// TwinCAT 3 PLC project Untitled1
// Title: B300S
// Company: LS do Brasil
// Author: Thiago Carlos
// ProjectVersion: 1.1
// Description: Programa da máquina B300S, 12 liquidos e dois pós
// ProgramVersion: 3.1.4024.0
// libraries:
//   Tc2_ControllerToolbox, * (Beckhoff Automation GmbH)
//   Tc2_Database, * (Beckhoff Automation GmbH)
//   Tc2_EtherCAT, * (Beckhoff Automation GmbH)
//   Tc2_Standard, * (Beckhoff Automation GmbH)
//   Tc2_System, * (Beckhoff Automation GmbH)
//   Tc2_Utilities, * (Beckhoff Automation GmbH)
//   Tc3_Database, * (Beckhoff Automation GmbH)
//   Tc3_EventLogger, * (Beckhoff Automation GmbH)
//   Tc3_IPCDiag, * (Beckhoff Automation GmbH)
//   Tc3_Module, * (Beckhoff Automation GmbH)
// project tree:
//   DUTs/ DUT_cfgBombas.TcDUT, DUT_cfgPosicValvula.TcDUT, DUT_PosicValvula.TcDUT, RecetaEdicion.TcDUT, stComboBoxRecipes.TcDUT, stListado_Liquidos.TcDUT, stListado_Polvos.TcDUT, stReceta_Circuito.TcDUT, stReceta_Polvo.TcDUT, u_RPM.TcDUT, u_SM6020.TcDUT, u_SM6020_caudal.TcDUT, u_SM6020_temp.TcDUT
//   / GVL.TcGVL, PlcTask.TcTTO
//   GVLs/ CanOpen.TcGVL, Configura.TcGVL, DatosProceso.TcGVL, Entradas.TcGVL, HMI.TcGVL, HMICA1.TcGVL, HMICA2.TcGVL, HMICA3.TcGVL, HMIcalP1.TcGVL, HMIcalP2.TcGVL, ioLink.TcGVL, Liquidos.TcGVL, Polvos.TcGVL, RecetasGestion.TcGVL, Receta_Activa.TcGVL, SafetyInputs.TcGVL, Salidas.TcGVL, Seguridad.TcGVL
//   POUs/ Agitadores.TcPOU, Alarmas.TcPOU, Balanza_Semilla.TcPOU, Datos_Caudalimetros.TcPOU, Datos_Variadores.TcPOU, Inicio.TcPOU, MAIN.TcPOU, PasosDosificar.TcPOU, PrecargaLiqInyeccion.TcPOU, Tabla_FIFO.TcPOU, VarPersistentes.TcPOU, Tratadora.TcPOU, _Seguridad.TcPOU
//   POUs/CanOpen/ SDO_READ.TcPOU
//   POUs/Control Equipos/ ControlValv_ioLink.TcPOU, Equipo_Motor_ATV320.TcPOU, Equipo_Motor_No_Rev.TcPOU, Equipo_Valvula_5_2.TcPOU, Equipo_Valvula_5_2_biestable.TcPOU
//   POUs/Elementos/ Calculo_caudal.TcPOU, Calc_Veloc_Polvo.TcPOU, Calibracion_Liq_calc.TcPOU, Calibracion_Po_calc.TcPOU, CorrecionCaudalxOffset.TcPOU, FB_PID.TcPOU, Tiempo_seg_to_TIME.TcPOU, Tiempo_TIME_to_seg.TcPOU
//   POUs/Lavado/ AbreValvulasLavagem.TcPOU, Valvulas_Lavado.TcPOU
//   POUs/Perifericos/ Carga_semilla.TcPOU, Descarga_semilla.TcPOU
//   POUs/Pesajes/ Balanza.TcPOU
//   POUs/Polvo 1/ Dosificador_Polvo_1.TcPOU
//   POUs/Polvo 2/ Dosificador_Polvo_2.TcPOU
//   POUs/Puesto_Calibracion_1/ Circuito_L1.TcPOU, Circuito_L2.TcPOU, Circuito_L3.TcPOU, Circuito_L4.TcPOU, Puesto_CA1.TcPOU
//   POUs/Puesto_Calibracion_2/ Circuito_L5.TcPOU, Circuito_L6.TcPOU, Circuito_L7.TcPOU, Circuito_L8.TcPOU, Puesto_CA2.TcPOU
//   POUs/Puesto_Calibracion_3/ Circuito_L11.TcPOU, Circuito_L12.TcPOU, Circuito_L9.TcPOU, Circuito_L10.TcPOU, Puesto_CA3.TcPOU
//   POUs/Receitas %28Thiago%29/ Receitas.TcPOU (not stored)
//   POUs/Secuencias/ Porc_inicial_Bomba.TcPOU, Totalizador.TcPOU, VeloAspersorAuto.TcPOU, LavadoCircuitoLiquidos.TcPOU
//   POUs/Testes Thiago/ AlarmesDaMaquina.TcPOU, AquecimentoValvulas.TcPOU, CalculoConsumo.TcPOU, Calibracao_V03.TcPOU, ConfigBombas.TcPOU, ConsumoIBCs.TcPOU, E_State.TcDUT, Filtro.TcPOU, Filtro2.TcPOU, GeraAlarme.TcPOU, BancoDeDados.TcPOU, Calibracao_V02.TcPOU, DUT_ConfigLavagem.TcDUT, DUT_EventLogger.TcDUT, InsertBD_Comandos.TcPOU, IntervaloLavCalibr.TcPOU, iPC_Diagnostic.TcPOU, Lavagem.TcPOU, LiqNaReceita.TcPOU, MediaMovel.TcPOU, Percentual.TcPOU, PRG_DE_TESTES.TcPOU, ST_SelectStruct.TcDUT, Testes.TcGVL, TONR.TcPOU
//   POUs/TestesPID/ PID_GENERICO.TcPOU
// real-time tasks:
//   TASK PlcTask: cycle T#10ms, priority 6, ADS port 352
// I/O:
//   DEVICE Dispositivos (EtherCAT) (disabled), AmsNetId 192.168.10.68.2.1
//     C1 (EK1100) [EK1100 EtherCAT Coupler (2A E-Bus)]
//       C2 (EL6070) [EL6070 1Ch. Licensing-Terminal]
//       C3 (EL1809) [EL1809 16Ch. Dig. Input 24V, 3ms]
//       C4 (EL2809) [EL2809 16Ch. Dig. Output 24V, 0.5A]
//       C6 (EL6224) [EL6224 (IO Link Master)]
//       C5 (EL2911) [EL2911, Potential supply terminal (10 A) with 4 Ch. Safety Inputs, TwinSAFE]
//         modules: Module 2 (FSOUT), Module 3 (DEVICEIO), Module 4 (FSLOGIC)
//       C7 (EL6753) [EL6751 CANopen Master]
//       C8 (EK1122) [EK1122 2 port EtherCAT junction]
//         CA1_1 (ifm IO-Link Master AL1332) [ifm IO-Link Master AL1332]
//           modules: Module 1 (IOL_16/4_I/O-Bytes), Module 2 (IOL_4/4_I/O-Bytes), Module 3 (IOL_16/4_I/O-Bytes), Module 4 (IOL_4/4_I/O-Bytes), Module 5 (IOL_16/4_I/O-Bytes), Module 6 (IOL_4/4_I/O-Bytes), Module 7 (IOL_16/4_I/O-Bytes), Module 8 (IOL_4/4_I/O-Bytes)
//         CA1_2 (EP3356-0022) [EP3356-0022 1Ch. Ana. Input Resistor Bridge Terminal, 24bit, High Precision]
//         PU1_1 (EP3356-0022) [EP3356-0022 1Ch. Ana. Input Resistor Bridge Terminal, 24bit, High Precision]
//         PU1_2 (ifm IO-Link Master AL1332) [ifm IO-Link Master AL1332]
//           modules: Module 1 (IOL_4/4_I/O-Bytes), Module 2 (IOL_4/4_I/O-Bytes), Module 3 (IOL_4/4_I/O-Bytes), Module 4 (IOL_4/4_I/O-Bytes), Module 5 (IOL_4/4_I/O-Bytes), Module 6 (IOL_4/4_I/O-Bytes), Module 7 (Digital_IN), Module 8 (Digital_IN)
//         PU1_3 (EP3356-0022) [EP3356-0022 1Ch. Ana. Input Resistor Bridge Terminal, 24bit, High Precision]
//         PU1_4 (EP3356-0022) [EP3356-0022 1Ch. Ana. Input Resistor Bridge Terminal, 24bit, High Precision]
//         PU1_5 (ifm IO-Link Master AL1332) [ifm IO-Link Master AL1332]
//           modules: Module 1 (IOL_4/4_I/O-Bytes), Module 2 (IOL_4/4_I/O-Bytes), Module 3 (IOL_4/4_I/O-Bytes), Module 4 (IOL_4/4_I/O-Bytes), Module 5 (IOL_4/4_I/O-Bytes), Module 6 (IOL_4/4_I/O-Bytes), Module 7 (Digital_IN), Module 8 (Digital_IN)
//         PU1_6 (EP3356-0022) [EP3356-0022 1Ch. Ana. Input Resistor Bridge Terminal, 24bit, High Precision]
//         PU4_1 (ifm IO-Link Master AL1330) [ifm IO-Link Master AL1330]
//           modules: Module 1 (IOL_4/4_I/O-Bytes), Module 2 (IOL_4/4_I/O-Bytes), Module 3 (IOL_4/4_I/O-Bytes), Module 4 (IOL_4/4_I/O-Bytes)
//         CA2_1 (ifm IO-Link Master AL1332) [ifm IO-Link Master AL1332]
//           modules: Module 1 (IOL_16/4_I/O-Bytes), Module 2 (IOL_4/4_I/O-Bytes), Module 3 (IOL_16/4_I/O-Bytes), Module 4 (IOL_4/4_I/O-Bytes), Module 5 (IOL_16/4_I/O-Bytes), Module 6 (IOL_4/4_I/O-Bytes), Module 7 (IOL_16/4_I/O-Bytes), Module 8 (IOL_4/4_I/O-Bytes)
//         CA2_2 (EP3356-0022) [EP3356-0022 1Ch. Ana. Input Resistor Bridge Terminal, 24bit, High Precision]
//         PU2_1 (EP3356-0022) [EP3356-0022 1Ch. Ana. Input Resistor Bridge Terminal, 24bit, High Precision]
//         PU2_2 (ifm IO-Link Master AL1332) [ifm IO-Link Master AL1332]
//           modules: Module 1 (IOL_4/4_I/O-Bytes), Module 2 (IOL_4/4_I/O-Bytes), Module 3 (IOL_4/4_I/O-Bytes), Module 4 (IOL_4/4_I/O-Bytes), Module 5 (IOL_4/4_I/O-Bytes), Module 6 (IOL_4/4_I/O-Bytes), Module 7 (Digital_IN), Module 8 (Digital_IN)
//         PU2_3 (EP3356-0022) [EP3356-0022 1Ch. Ana. Input Resistor Bridge Terminal, 24bit, High Precision]
//         PU2_4 (EP3356-0022) [EP3356-0022 1Ch. Ana. Input Resistor Bridge Terminal, 24bit, High Precision]
//         PU2_5 (ifm IO-Link Master AL1332) [ifm IO-Link Master AL1332]
//           modules: Module 1 (IOL_4/4_I/O-Bytes), Module 2 (IOL_4/4_I/O-Bytes), Module 3 (IOL_4/4_I/O-Bytes), Module 4 (IOL_4/4_I/O-Bytes), Module 5 (IOL_4/4_I/O-Bytes), Module 6 (IOL_4/4_I/O-Bytes), Module 7 (Digital_IN), Module 8 (Digital_IN)
//         PU2_6 (EP3356-0022) [EP3356-0022 1Ch. Ana. Input Resistor Bridge Terminal, 24bit, High Precision]
//       C9 (EK1122) [EK1122 2 port EtherCAT junction]
//         CA3_1 (ifm IO-Link Master AL1332) [ifm IO-Link Master AL1332]
//           modules: Module 1 (IOL_16/4_I/O-Bytes), Module 2 (IOL_4/4_I/O-Bytes), Module 3 (IOL_16/4_I/O-Bytes), Module 4 (IOL_4/4_I/O-Bytes), Module 5 (IOL_16/4_I/O-Bytes), Module 6 (IOL_4/4_I/O-Bytes), Module 7 (IOL_16/4_I/O-Bytes), Module 8 (IOL_4/4_I/O-Bytes)
//         CA3_2 (EP3356-0022) [EP3356-0022 1Ch. Ana. Input Resistor Bridge Terminal, 24bit, High Precision]
//         PU3_1 (EP3356-0022) [EP3356-0022 1Ch. Ana. Input Resistor Bridge Terminal, 24bit, High Precision]
//         PU3_2 (ifm IO-Link Master AL1332) [ifm IO-Link Master AL1332]
//           modules: Module 1 (IOL_4/4_I/O-Bytes), Module 2 (IOL_4/4_I/O-Bytes), Module 3 (IOL_4/4_I/O-Bytes), Module 4 (IOL_4/4_I/O-Bytes), Module 5 (IOL_4/4_I/O-Bytes), Module 6 (IOL_4/4_I/O-Bytes), Module 7 (Digital_IN), Module 8 (Digital_IN)
//         PU3_3 (EP3356-0022) [EP3356-0022 1Ch. Ana. Input Resistor Bridge Terminal, 24bit, High Precision]
//         PU3_4 (EP3356-0022) [EP3356-0022 1Ch. Ana. Input Resistor Bridge Terminal, 24bit, High Precision]
//         PU3_5 (ifm IO-Link Master AL1332) [ifm IO-Link Master AL1332]
//           modules: Module 1 (IOL_4/4_I/O-Bytes), Module 2 (IOL_4/4_I/O-Bytes), Module 3 (IOL_4/4_I/O-Bytes), Module 4 (IOL_4/4_I/O-Bytes), Module 5 (IOL_4/4_I/O-Bytes), Module 6 (IOL_4/4_I/O-Bytes), Module 7 (Digital_IN), Module 8 (Digital_IN)
//         PU3_6 (EP3356-0022) [EP3356-0022 1Ch. Ana. Input Resistor Bridge Terminal, 24bit, High Precision]
//         PE_2 (ifm IO-Link Master AL1332) [ifm IO-Link Master AL1332]
//           modules: Module 1 (IOL_4/4_I/O-Bytes), Module 2 (IOL_4/4_I/O-Bytes), Module 3 (IOL_4/4_I/O-Bytes), Module 4 (IOL_4/4_I/O-Bytes), Module 5 (IOL_4/4_I/O-Bytes), Module 6 (IOL_4/4_I/O-Bytes), Module 7 (IOL_4/4_I/O-Bytes), Module 8 (IOL_4/4_I/O-Bytes)
//         PE_1 (EX260-SEC1) [EX260-SEC1 EtherCAT SI Unit (32DO_PNP) Rev1.2]
//         PE_4 (ifm IO-Link Master AL1330) [ifm IO-Link Master AL1330]
//           modules: Module 1 (IOL_4/4_I/O-Bytes), Module 2 (Digital_IN), Module 3 (Digital_IN), Module 4 (Digital_IN)
//         PE_3 (EX260-SEC1) [EX260-SEC1 EtherCAT SI Unit (32DO_PNP) Rev1.2]
//         Box 37 (EX260-SEC1) [EX260-SEC1 EtherCAT SI Unit (32DO_PNP) Rev1.2] (disabled)
//     TR_1 (EP3356-0022) [EP3356-0022 1Ch. Ana. Input Resistor Bridge Terminal, 24bit, High Precision]
//     TR_2 (EP1908) [EP1908, 8 Ch. Safety Input 24V, TwinSAFE ]
//       modules: Module 1 (FSOE)
//     TR_3 (EP1908) [EP1908, 8 Ch. Safety Input 24V, TwinSAFE ]
//       modules: Module 1 (FSOE)
//     TR_4 (ifm IO-Link Master AL1332) [ifm IO-Link Master AL1332]
//       modules: Module 1 (Digital_IN), Module 2 (Digital_IN), Module 3 (Digital_IN), Module 4 (Digital_IN), Module 5 (Digital_IN), Module 6 (Digital_IN), Module 7 (IOL_In_4Byte), Module 8 (IOL_In_4Byte)
//     TR_5 (EX260-SEC1) [EX260-SEC1 EtherCAT SI Unit (32DO_PNP) Rev1.2]
//     TR_6 (ifm IO-Link Master AL1332) [ifm IO-Link Master AL1332]
//       modules: Module 1 (IOL_16/4_I/O-Bytes), Module 2 (IOL_16/4_I/O-Bytes), Module 3 (IOL_16/4_I/O-Bytes), Module 4 (IOL_16/4_I/O-Bytes), Module 5 (IOL_16/4_I/O-Bytes), Module 6 (IOL_16/4_I/O-Bytes), Module 7 (IOL_16/4_I/O-Bytes), Module 8 (IOL_16/4_I/O-Bytes)
//     TR_7 (ifm IO-Link Master AL1330) [ifm IO-Link Master AL1330]
//       modules: Module 1 (IOL_16/4_I/O-Bytes), Module 2 (IOL_16/4_I/O-Bytes), Module 3 (IOL_16/4_I/O-Bytes), Module 4 (IOL_16/4_I/O-Bytes)
//     TR_8 (ifm IO-Link Master AL1332) [ifm IO-Link Master AL1332]
//       modules: Module 1 (IOL_4/4_I/O-Bytes), Module 2 (IOL_4/4_I/O-Bytes), Module 3 (Digital_IN), Module 4 (Digital_IN), Module 5 (Digital_IN), Module 6 (Digital_OUT), Module 7 (IOL_4/4_I/O-Bytes), Module 8 (IOL_4/4_I/O-Bytes)
//     TR_9 (ifm IO-Link Master AL1330) [ifm IO-Link Master AL1330]
//       modules: Module 1 (Digital_IN), Module 2 (Digital_IN), Module 3 (Digital_IN), Module 4 (IOL_4/4_I/O-Bytes)
//     TR_10 (EP3356-0022) [EP3356-0022 1Ch. Ana. Input Resistor Bridge Terminal, 24bit, High Precision]
//     TR_11 (ifm IO-Link Master AL1330) [ifm IO-Link Master AL1330]
//       modules: Module 1 (Digital_IN), Module 2 (Digital_IN), Module 3 (Digital_IN), Module 4 (Digital_IN)
//     TR_12 (EP3356-0022) [EP3356-0022 1Ch. Ana. Input Resistor Bridge Terminal, 24bit, High Precision]
//   DEVICE Device 2 (EL6751), AmsNetId 169.254.25.50.4.1
//     Box 1 (ATV320D15N4C)
//     Box 2 (ATV320U07M2C)
//     Box 3 (ATV320U06M2C)
//     Box 4 (ATV320U06M2C)
//     Box 5 (ATV320U07M2C)
//     Box 6 (ATV320U04M2C)
//     Box 7 (ATV320U04M2C)
//     Box 8 (ATV320U04M2C)
//     Box 9 (ATV320U04M2C)
//     Box 10 (ATV320U04M2C)
//     Box 11 (ATV320U04M2C)
//     Box 12 (ATV320U04M2C)
//     Box 13 (ATV320U04M2C)
//     Box 14 (ATV320U04M2C)
//     Box 15 (ATV320U04M2C)
//     Box 16 (ATV320U04M2C)
//     Box 17 (ATV320U15M2C)
//     Box 18 (ATV320U15M2C)
//     Box 19 (ATV320U22M2C)
//     Box 34 (ATV320U04M2C)
//     Box 35 (ATV320U04M2C)
// variable links:
//   Dispositivos (EtherCAT) <-> Dispositivos (EtherCAT)/C1 (EK1100)/C5 (EL2911)
//     TR_2 (EP1908)/Module 1 (FSOE)/FSOE Outputs/FSOE <-> ConnectionInputs/Message_18 TxPDO
//   Dispositivos (EtherCAT) <-> Dispositivos (EtherCAT)/TR_2 (EP1908)
//     C1 (EK1100)/C5 (EL2911)/ConnectionOutputs/Message_18 RxPDO <-> Module 1 (FSOE)/FSOE Inputs/FSOE
//   Dispositivos (EtherCAT) <-> Dispositivos (EtherCAT)/TR_3 (EP1908)
//     C1 (EK1100)/C5 (EL2911)/ConnectionInputs/Message_19 TxPDO <-> Module 1 (FSOE)/FSOE Outputs/FSOE
//     C1 (EK1100)/C5 (EL2911)/ConnectionOutputs/Message_19 RxPDO <-> Module 1 (FSOE)/FSOE Inputs/FSOE
//   Untitled1/Untitled1 Instance <-> Device 2 (EL6751)/Box 1 (ATV320D15N4C)
//     PlcTask Inputs/Entradas.wTR_S_VF1_PV <-> TxPDO 1/Inputs/VarIn-1
//     PlcTask Inputs/Entradas.wTR_S_VF1_St <-> TxPDO 1/Inputs/VarIn-0
//     PlcTask Outputs/Salidas.wTR_S_VF1_Cmd <-> RxPDO 1/Outputs/VarOut-0
//     PlcTask Outputs/Salidas.wTR_S_VF1_Set <-> RxPDO 1/Outputs/VarOut-1
//   Untitled1/Untitled1 Instance <-> Device 2 (EL6751)/Box 10 (ATV320U04M2C)
//     PlcTask Inputs/Entradas.wPP2_L6_BD_PV <-> TxPDO 1/Inputs/VarIn-1
//     PlcTask Inputs/Entradas.wPP2_L6_BD_St <-> TxPDO 1/Inputs/VarIn-0
//     PlcTask Outputs/Salidas.wPP2_L6_BD_Cmd <-> RxPDO 1/Outputs/VarOut-0
//     PlcTask Outputs/Salidas.wPP2_L6_BD_Set <-> RxPDO 1/Outputs/VarOut-1
//   Untitled1/Untitled1 Instance <-> Device 2 (EL6751)/Box 11 (ATV320U04M2C)
//     PlcTask Inputs/Entradas.wPP2_L7_BD_PV <-> TxPDO 1/Inputs/VarIn-1
//     PlcTask Inputs/Entradas.wPP2_L7_BD_St <-> TxPDO 1/Inputs/VarIn-0
//     PlcTask Outputs/Salidas.wPP2_L7_BD_Cmd <-> RxPDO 1/Outputs/VarOut-0
//     PlcTask Outputs/Salidas.wPP2_L7_BD_Set <-> RxPDO 1/Outputs/VarOut-1
//   Untitled1/Untitled1 Instance <-> Device 2 (EL6751)/Box 12 (ATV320U04M2C)
//     PlcTask Inputs/Entradas.wPP2_L8_BD_PV <-> TxPDO 1/Inputs/VarIn-1
//     PlcTask Inputs/Entradas.wPP2_L8_BD_St <-> TxPDO 1/Inputs/VarIn-0
//     PlcTask Outputs/Salidas.wPP2_L8_BD_Cmd <-> RxPDO 1/Outputs/VarOut-0
//     PlcTask Outputs/Salidas.wPP2_L8_BD_Set <-> RxPDO 1/Outputs/VarOut-1
//   Untitled1/Untitled1 Instance <-> Device 2 (EL6751)/Box 13 (ATV320U04M2C)
//     PlcTask Inputs/Entradas.wPP3_L9_BD_PV <-> TxPDO 1/Inputs/VarIn-1
//     PlcTask Inputs/Entradas.wPP3_L9_BD_St <-> TxPDO 1/Inputs/VarIn-0
//     PlcTask Outputs/Salidas.wPP3_L9_BD_Cmd <-> RxPDO 1/Outputs/VarOut-0
//     PlcTask Outputs/Salidas.wPP3_L9_BD_Set <-> RxPDO 1/Outputs/VarOut-1
//   Untitled1/Untitled1 Instance <-> Device 2 (EL6751)/Box 14 (ATV320U04M2C)
//     PlcTask Inputs/Entradas.wPP3_L10_BD_PV <-> TxPDO 1/Inputs/VarIn-1
//     PlcTask Inputs/Entradas.wPP3_L10_BD_St <-> TxPDO 1/Inputs/VarIn-0
//     PlcTask Outputs/Salidas.wPP3_L10_BD_Cmd <-> RxPDO 1/Outputs/VarOut-0
//     PlcTask Outputs/Salidas.wPP3_L10_BD_Set <-> RxPDO 1/Outputs/VarOut-1
//   Untitled1/Untitled1 Instance <-> Device 2 (EL6751)/Box 15 (ATV320U04M2C)
//     PlcTask Inputs/Entradas.wPP3_L11_BD_PV <-> TxPDO 1/Inputs/VarIn-1
//     PlcTask Inputs/Entradas.wPP3_L11_BD_St <-> TxPDO 1/Inputs/VarIn-0
//     PlcTask Outputs/Salidas.wPP3_L11_BD_Cmd <-> RxPDO 1/Outputs/VarOut-0
//     PlcTask Outputs/Salidas.wPP3_L11_BD_Set <-> RxPDO 1/Outputs/VarOut-1
//   Untitled1/Untitled1 Instance <-> Device 2 (EL6751)/Box 16 (ATV320U04M2C)
//     PlcTask Inputs/Entradas.wPP3_L12_BD_PV <-> TxPDO 1/Inputs/VarIn-1
//     PlcTask Inputs/Entradas.wPP3_L12_BD_St <-> TxPDO 1/Inputs/VarIn-0
//     PlcTask Outputs/Salidas.wPP3_L12_BD_Cmd <-> RxPDO 1/Outputs/VarOut-0
//     PlcTask Outputs/Salidas.wPP3_L12_BD_Set <-> RxPDO 1/Outputs/VarOut-1
//   Untitled1/Untitled1 Instance <-> Device 2 (EL6751)/Box 17 (ATV320U15M2C)
//     PlcTask Inputs/Entradas.wPE_H_VF1_PV <-> TxPDO 1/Inputs/VarIn-1
//     PlcTask Inputs/Entradas.wPE_H_VF1_St <-> TxPDO 1/Inputs/VarIn-0
//     PlcTask Outputs/Salidas.wPE_H_VF1_Cmd <-> RxPDO 1/Outputs/VarOut-0
//     PlcTask Outputs/Salidas.wPE_H_VF1_Set <-> RxPDO 1/Outputs/VarOut-1
//   Untitled1/Untitled1 Instance <-> Device 2 (EL6751)/Box 18 (ATV320U15M2C)
//     PlcTask Inputs/Entradas.wPE_H_VF2_PV <-> TxPDO 1/Inputs/VarIn-1
//     PlcTask Inputs/Entradas.wPE_H_VF2_St <-> TxPDO 1/Inputs/VarIn-0
//     PlcTask Outputs/Salidas.wPE_H_VF2_Cmd <-> RxPDO 1/Outputs/VarOut-0
//     PlcTask Outputs/Salidas.wPE_H_VF2_Set <-> RxPDO 1/Outputs/VarOut-1
//   Untitled1/Untitled1 Instance <-> Device 2 (EL6751)/Box 19 (ATV320U22M2C)
//     PlcTask Inputs/Entradas.wPE_B_VF1_PV <-> TxPDO 1/Inputs/VarIn-1
//     PlcTask Inputs/Entradas.wPE_B_VF1_St <-> TxPDO 1/Inputs/VarIn-0
//     PlcTask Outputs/Salidas.wPE_B_VF1_Cmd <-> RxPDO 1/Outputs/VarOut-0
//     PlcTask Outputs/Salidas.wPE_B_VF1_Set <-> RxPDO 1/Outputs/VarOut-1
//   Untitled1/Untitled1 Instance <-> Device 2 (EL6751)/Box 2 (ATV320U07M2C)
//     PlcTask Inputs/Entradas.wTR_S_VF2_PV <-> TxPDO 1/Inputs/VarIn-1
//     PlcTask Inputs/Entradas.wTR_S_VF2_St <-> TxPDO 1/Inputs/VarIn-0
//     PlcTask Outputs/Salidas.wTR_S_VF2_Cmd <-> RxPDO 1/Outputs/VarOut-0
//     PlcTask Outputs/Salidas.wTR_S_VF2_Set <-> RxPDO 1/Outputs/VarOut-1
//   Untitled1/Untitled1 Instance <-> Device 2 (EL6751)/Box 3 (ATV320U06M2C)
//     PlcTask Inputs/Entradas.TR_P1_VF_PV <-> TxPDO 1/Inputs/VarIn-1
//     PlcTask Inputs/Entradas.TR_P1_VF_St <-> TxPDO 1/Inputs/VarIn-0
//     PlcTask Outputs/Salidas.TR_P1_VF_Cmd <-> RxPDO 1/Outputs/VarOut-0
//     PlcTask Outputs/Salidas.TR_P1_VF_Set <-> RxPDO 1/Outputs/VarOut-1
//   Untitled1/Untitled1 Instance <-> Device 2 (EL6751)/Box 34 (ATV320U04M2C)
//     PlcTask Inputs/Entradas.TR_P1_VI_PV <-> TxPDO 1/Inputs/VarIn-1
//     PlcTask Inputs/Entradas.TR_P1_VI_St <-> TxPDO 1/Inputs/VarIn-0
//     PlcTask Outputs/Salidas.TR_P1_VI_Cmd <-> RxPDO 1/Outputs/VarOut-0
//     PlcTask Outputs/Salidas.TR_P1_VI_Set <-> RxPDO 1/Outputs/VarOut-1
//   Untitled1/Untitled1 Instance <-> Device 2 (EL6751)/Box 35 (ATV320U04M2C)
//     PlcTask Inputs/Entradas.TR_P2_VI_PV <-> TxPDO 1/Inputs/VarIn-1
//     PlcTask Inputs/Entradas.TR_P2_VI_St <-> TxPDO 1/Inputs/VarIn-0
//     PlcTask Outputs/Salidas.TR_P2_VI_Cmd <-> RxPDO 1/Outputs/VarOut-0
//     PlcTask Outputs/Salidas.TR_P2_VI_Set <-> RxPDO 1/Outputs/VarOut-1
//   Untitled1/Untitled1 Instance <-> Device 2 (EL6751)/Box 4 (ATV320U06M2C)
//     PlcTask Inputs/Entradas.TR_P2_VF_PV <-> TxPDO 1/Inputs/VarIn-1
//     PlcTask Inputs/Entradas.TR_P2_VF_St <-> TxPDO 1/Inputs/VarIn-0
//     PlcTask Outputs/Salidas.TR_P2_VF_Cmd <-> RxPDO 1/Outputs/VarOut-0
//     PlcTask Outputs/Salidas.TR_P2_VF_Set <-> RxPDO 1/Outputs/VarOut-1
//   Untitled1/Untitled1 Instance <-> Device 2 (EL6751)/Box 5 (ATV320U07M2C)
//     PlcTask Inputs/Entradas.wPP1_L1_BD_PV <-> TxPDO 1/Inputs/VarIn-1
//     PlcTask Inputs/Entradas.wPP1_L1_BD_St <-> TxPDO 1/Inputs/VarIn-0
//     PlcTask Outputs/Salidas.wPP1_L1_BD_Cmd <-> RxPDO 1/Outputs/VarOut-0
//     PlcTask Outputs/Salidas.wPP1_L1_BD_Set <-> RxPDO 1/Outputs/VarOut-1
//   Untitled1/Untitled1 Instance <-> Device 2 (EL6751)/Box 6 (ATV320U04M2C)
//     PlcTask Inputs/Entradas.wPP1_L2_BD_PV <-> TxPDO 1/Inputs/VarIn-1
//     PlcTask Inputs/Entradas.wPP1_L2_BD_St <-> TxPDO 1/Inputs/VarIn-0
//     PlcTask Outputs/Salidas.wPP1_L2_BD_Cmd <-> RxPDO 1/Outputs/VarOut-0
//     PlcTask Outputs/Salidas.wPP1_L2_BD_Set <-> RxPDO 1/Outputs/VarOut-1
//   Untitled1/Untitled1 Instance <-> Device 2 (EL6751)/Box 7 (ATV320U04M2C)
//     PlcTask Inputs/Entradas.wPP1_L3_BD_PV <-> TxPDO 1/Inputs/VarIn-1
//     PlcTask Inputs/Entradas.wPP1_L3_BD_St <-> TxPDO 1/Inputs/VarIn-0
//     PlcTask Outputs/Salidas.wPP1_L3_BD_Cmd <-> RxPDO 1/Outputs/VarOut-0
//     PlcTask Outputs/Salidas.wPP1_L3_BD_Set <-> RxPDO 1/Outputs/VarOut-1
//   Untitled1/Untitled1 Instance <-> Device 2 (EL6751)/Box 8 (ATV320U04M2C)
//     PlcTask Inputs/Entradas.wPP1_L4_BD_PV <-> TxPDO 1/Inputs/VarIn-1
//     PlcTask Inputs/Entradas.wPP1_L4_BD_St <-> TxPDO 1/Inputs/VarIn-0
//     PlcTask Outputs/Salidas.wPP1_L4_BD_Cmd <-> RxPDO 1/Outputs/VarOut-0
//     PlcTask Outputs/Salidas.wPP1_L4_BD_Set <-> RxPDO 1/Outputs/VarOut-1
//   Untitled1/Untitled1 Instance <-> Device 2 (EL6751)/Box 9 (ATV320U04M2C)
//     PlcTask Inputs/Entradas.wPP2_L5_BD_PV <-> TxPDO 1/Inputs/VarIn-1
//     PlcTask Inputs/Entradas.wPP2_L5_BD_St <-> TxPDO 1/Inputs/VarIn-0
//     PlcTask Outputs/Salidas.wPP2_L5_BD_Cmd <-> RxPDO 1/Outputs/VarOut-0
//     PlcTask Outputs/Salidas.wPP2_L5_BD_Set <-> RxPDO 1/Outputs/VarOut-1
//   Untitled1/Untitled1 Instance <-> Dispositivos (EtherCAT)/C1 (EK1100)/C3 (EL1809)
//     PlcTask Inputs/Entradas.ReposicionEmerg <-> Channel 15/Input
//     PlcTask Inputs/Entradas.bPP1_L1_AG_Z <-> Channel 2/Input
//     PlcTask Inputs/Entradas.bPP1_L2_AG_Z <-> Channel 3/Input
//     PlcTask Inputs/Entradas.bPP1_L3_AG_Z <-> Channel 4/Input
//     PlcTask Inputs/Entradas.bPP1_L4_AG_Z <-> Channel 5/Input
//     PlcTask Inputs/Entradas.bPP2_L5_AG_Z <-> Channel 6/Input
//     PlcTask Inputs/Entradas.bPP2_L6_AG_Z <-> Channel 7/Input
//     PlcTask Inputs/Entradas.bPP2_L7_AG_Z <-> Channel 8/Input
//     PlcTask Inputs/Entradas.bPP2_L8_AG_Z <-> Channel 9/Input
//     PlcTask Inputs/Entradas.bPP3_L10_AG_Z <-> Channel 11/Input
//     PlcTask Inputs/Entradas.bPP3_L11_AG_Z <-> Channel 12/Input
//     PlcTask Inputs/Entradas.bPP3_L12_AG_Z <-> Channel 13/Input
//     PlcTask Inputs/Entradas.bPP3_L9_AG_Z <-> Channel 10/Input
//     PlcTask Inputs/Entradas.bTR_S_VE1_Z <-> Channel 1/Input
//   Untitled1/Untitled1 Instance <-> Dispositivos (EtherCAT)/C1 (EK1100)/C4 (EL2809)
//     PlcTask Outputs/Salidas.PE_P1_HC <-> Channel 14/Output
//     PlcTask Outputs/Salidas.PE_P2_HC <-> Channel 16/Output
//     PlcTask Outputs/Salidas.bPP1_L1_AG_M <-> Channel 2/Output
//     PlcTask Outputs/Salidas.bPP1_L2_AG_M <-> Channel 3/Output
//     PlcTask Outputs/Salidas.bPP1_L3_AG_M <-> Channel 4/Output
//     PlcTask Outputs/Salidas.bPP1_L4_AG_M <-> Channel 5/Output
//     PlcTask Outputs/Salidas.bPP2_L5_AG_M <-> Channel 6/Output
//     PlcTask Outputs/Salidas.bPP2_L6_AG_M <-> Channel 7/Output
//     PlcTask Outputs/Salidas.bPP2_L7_AG_M <-> Channel 8/Output
//     PlcTask Outputs/Salidas.bPP2_L8_AG_M <-> Channel 9/Output
//     PlcTask Outputs/Salidas.bPP3_L10_AG_M <-> Channel 11/Output
//     PlcTask Outputs/Salidas.bPP3_L11_AG_M <-> Channel 12/Output
//     PlcTask Outputs/Salidas.bPP3_L12_AG_M <-> Channel 13/Output
//     PlcTask Outputs/Salidas.bPP3_L9_AG_M <-> Channel 10/Output
//     PlcTask Outputs/Salidas.bTR_S_VE1 <-> Channel 1/Output
//   Untitled1/Untitled1 Instance <-> Dispositivos (EtherCAT)/C1 (EK1100)/C5 (EL2911)
//     PlcTask Inputs/Seguridad.PB_Emergencia <-> StandardInputs/Standard Out Var 8
//     PlcTask Inputs/Seguridad.ParadaDePorta <-> StandardInputs/Standard Out Var 12
//     PlcTask Outputs/Seguridad.ErrorAck <-> StandardOutputs/Standard In Var 1
//     PlcTask Outputs/Seguridad.ResetPorta <-> StandardOutputs/Standard In Var 14
//     PlcTask Outputs/Seguridad.Restart <-> StandardOutputs/Standard In Var 4
//     PlcTask Outputs/Seguridad.Run <-> StandardOutputs/Standard In Var 2
//   Untitled1/Untitled1 Instance <-> Dispositivos (EtherCAT)/C1 (EK1100)/C8 (EK1122)/CA1_1 (ifm IO-Link Master AL1332)
//     PlcTask Inputs/Entradas.CA1_L1_FT1_caudal/caudal[0] <-> Module 1 (IOL_16/4_I/O-Bytes)/TxPDO/input byte 5
//     PlcTask Inputs/Entradas.CA1_L1_FT1_caudal/caudal[1] <-> Module 1 (IOL_16/4_I/O-Bytes)/TxPDO/input byte 4
//     PlcTask Inputs/Entradas.CA1_L2_FT1_caudal/caudal[0] <-> Module 3 (IOL_16/4_I/O-Bytes)/TxPDO/input byte 5
//     PlcTask Inputs/Entradas.CA1_L2_FT1_caudal/caudal[1] <-> Module 3 (IOL_16/4_I/O-Bytes)/TxPDO/input byte 4
//     PlcTask Inputs/Entradas.CA1_L3_FT1_caudal/caudal[0] <-> Module 5 (IOL_16/4_I/O-Bytes)/TxPDO/input byte 5
//     PlcTask Inputs/Entradas.CA1_L3_FT1_caudal/caudal[1] <-> Module 5 (IOL_16/4_I/O-Bytes)/TxPDO/input byte 4
//     PlcTask Inputs/Entradas.CA1_L4_FT1_caudal/caudal[0] <-> Module 7 (IOL_16/4_I/O-Bytes)/TxPDO/input byte 5
//     PlcTask Inputs/Entradas.CA1_L4_FT1_caudal/caudal[1] <-> Module 7 (IOL_16/4_I/O-Bytes)/TxPDO/input byte 4
//     PlcTask Inputs/Entradas.CA1_L1_FT1_temp/temp[0] <-> Module 1 (IOL_16/4_I/O-Bytes)/TxPDO/input byte 9
//     PlcTask Inputs/Entradas.CA1_L1_FT1_temp/temp[1] <-> Module 1 (IOL_16/4_I/O-Bytes)/TxPDO/input byte 8
//     PlcTask Inputs/Entradas.CA1_L2_FT1_temp/temp[0] <-> Module 3 (IOL_16/4_I/O-Bytes)/TxPDO/input byte 9
//     PlcTask Inputs/Entradas.CA1_L2_FT1_temp/temp[1] <-> Module 3 (IOL_16/4_I/O-Bytes)/TxPDO/input byte 8
//     PlcTask Inputs/Entradas.CA1_L3_FT1_temp/temp[0] <-> Module 5 (IOL_16/4_I/O-Bytes)/TxPDO/input byte 9
//     PlcTask Inputs/Entradas.CA1_L3_FT1_temp/temp[1] <-> Module 5 (IOL_16/4_I/O-Bytes)/TxPDO/input byte 8
//     PlcTask Inputs/Entradas.CA1_L4_FT1_temp/temp[0] <-> Module 7 (IOL_16/4_I/O-Bytes)/TxPDO/input byte 9
//     PlcTask Inputs/Entradas.CA1_L4_FT1_temp/temp[1] <-> Module 7 (IOL_16/4_I/O-Bytes)/TxPDO/input byte 8
//     PlcTask Inputs/Entradas.CA1_L1_FT1_tot/total[0] <-> Module 1 (IOL_16/4_I/O-Bytes)/TxPDO/input byte 3
//     PlcTask Inputs/Entradas.CA1_L1_FT1_tot/total[1] <-> Module 1 (IOL_16/4_I/O-Bytes)/TxPDO/input byte 2
//     PlcTask Inputs/Entradas.CA1_L1_FT1_tot/total[2] <-> Module 1 (IOL_16/4_I/O-Bytes)/TxPDO/input byte 1
//     PlcTask Inputs/Entradas.CA1_L1_FT1_tot/total[3] <-> Module 1 (IOL_16/4_I/O-Bytes)/TxPDO/input byte 0
//     PlcTask Inputs/Entradas.CA1_L2_FT1_tot/total[0] <-> Module 3 (IOL_16/4_I/O-Bytes)/TxPDO/input byte 3
//     PlcTask Inputs/Entradas.CA1_L2_FT1_tot/total[1] <-> Module 3 (IOL_16/4_I/O-Bytes)/TxPDO/input byte 2
//     PlcTask Inputs/Entradas.CA1_L2_FT1_tot/total[2] <-> Module 3 (IOL_16/4_I/O-Bytes)/TxPDO/input byte 1
//     PlcTask Inputs/Entradas.CA1_L2_FT1_tot/total[3] <-> Module 3 (IOL_16/4_I/O-Bytes)/TxPDO/input byte 0
//     PlcTask Inputs/Entradas.CA1_L4_FT1_tot/total[0] <-> Module 7 (IOL_16/4_I/O-Bytes)/TxPDO/input byte 3
//     PlcTask Inputs/Entradas.CA1_L4_FT1_tot/total[1] <-> Module 7 (IOL_16/4_I/O-Bytes)/TxPDO/input byte 2
//     PlcTask Inputs/Entradas.CA1_L4_FT1_tot/total[2] <-> Module 7 (IOL_16/4_I/O-Bytes)/TxPDO/input byte 1
//     PlcTask Inputs/Entradas.CA1_L4_FT1_tot/total[3] <-> Module 7 (IOL_16/4_I/O-Bytes)/TxPDO/input byte 0
//     PlcTask Inputs/Entradas.CA1_L1_V1_POSIC/Posicao[0] <-> Module 2 (IOL_4/4_I/O-Bytes)/TxPDO/input byte 0
//     PlcTask Inputs/Entradas.CA1_L1_V1_POSIC/Posicao[1] <-> Module 2 (IOL_4/4_I/O-Bytes)/TxPDO/input byte 1
//     PlcTask Inputs/Entradas.CA1_L2_V1_POSIC/Posicao[0] <-> Module 4 (IOL_4/4_I/O-Bytes)/TxPDO/input byte 0
//     PlcTask Inputs/Entradas.CA1_L2_V1_POSIC/Posicao[1] <-> Module 4 (IOL_4/4_I/O-Bytes)/TxPDO/input byte 1
//     PlcTask Inputs/Entradas.CA1_L3_V1_POSIC/Posicao[0] <-> Module 6 (IOL_4/4_I/O-Bytes)/TxPDO/input byte 0
//     PlcTask Inputs/Entradas.CA1_L3_V1_POSIC/Posicao[1] <-> Module 6 (IOL_4/4_I/O-Bytes)/TxPDO/input byte 1
//     PlcTask Inputs/Entradas.CA1_L4_V1_POSIC/Posicao[0] <-> Module 8 (IOL_4/4_I/O-Bytes)/TxPDO/input byte 0
//     PlcTask Inputs/Entradas.CA1_L4_V1_POSIC/Posicao[1] <-> Module 8 (IOL_4/4_I/O-Bytes)/TxPDO/input byte 1
//     PlcTask Inputs/Entradas.CA1_L3_FT1_Tot/total[{0..3}] <-> Module 5 (IOL_16/4_I/O-Bytes)/TxPDO/input byte {3..0}  (4 links)
//     PlcTask Inputs/ioLink.b3St1_CA1_L{1..4}_V1 <-> Module {2..8 step 2} (IOL_4/4_I/O-Bytes)/TxPDO/input byte 3  (4 links)
//     PlcTask Outputs/ioLink.b0Cmd_CA1_L{1..4}_V1 <-> Module {2..8 step 2} (IOL_4/4_I/O-Bytes)/RxPDO/output byte 0  (4 links)
//   Untitled1/Untitled1 Instance <-> Dispositivos (EtherCAT)/C1 (EK1100)/C8 (EK1122)/CA1_2 (EP3356-0022)
//     PlcTask Inputs/Entradas.CA1_WT1_bWcState <-> WcState/WcState
//     PlcTask Inputs/Entradas.CA1_WT1_rValue_REAL <-> RMB Value (Real)/Value (Real)
//     PlcTask Inputs/Entradas.CA1_WT1_stEcSlaveAmsNetAdr <-> InfoData/AdsAddr
//     PlcTask Inputs/Entradas.CA1_WT1_wState <-> InfoData/State
//     PlcTask Inputs/Entradas.CA1_WT1_wStatus <-> RMB Status/Status
//     PlcTask Outputs/Salidas.CA1_WT1_wControl <-> RMB Control/Ctrl
//   Untitled1/Untitled1 Instance <-> Dispositivos (EtherCAT)/C1 (EK1100)/C8 (EK1122)/CA2_1 (ifm IO-Link Master AL1332)
//     PlcTask Inputs/Entradas.CA2_L5_FT1_caudal/caudal[0] <-> Module 1 (IOL_16/4_I/O-Bytes)/TxPDO/input byte 5
//     PlcTask Inputs/Entradas.CA2_L5_FT1_caudal/caudal[1] <-> Module 1 (IOL_16/4_I/O-Bytes)/TxPDO/input byte 4
//     PlcTask Inputs/Entradas.CA2_L6_FT1_caudal/caudal[0] <-> Module 3 (IOL_16/4_I/O-Bytes)/TxPDO/input byte 5
//     PlcTask Inputs/Entradas.CA2_L6_FT1_caudal/caudal[1] <-> Module 3 (IOL_16/4_I/O-Bytes)/TxPDO/input byte 4
//     PlcTask Inputs/Entradas.CA2_L7_FT1_caudal/caudal[0] <-> Module 5 (IOL_16/4_I/O-Bytes)/TxPDO/input byte 5
//     PlcTask Inputs/Entradas.CA2_L7_FT1_caudal/caudal[1] <-> Module 5 (IOL_16/4_I/O-Bytes)/TxPDO/input byte 4
//     PlcTask Inputs/Entradas.CA2_L8_FT1_caudal/caudal[0] <-> Module 7 (IOL_16/4_I/O-Bytes)/TxPDO/input byte 5
//     PlcTask Inputs/Entradas.CA2_L8_FT1_caudal/caudal[1] <-> Module 7 (IOL_16/4_I/O-Bytes)/TxPDO/input byte 4
//     PlcTask Inputs/Entradas.CA2_L5_FT1_temp/temp[0] <-> Module 1 (IOL_16/4_I/O-Bytes)/TxPDO/input byte 9
//     PlcTask Inputs/Entradas.CA2_L5_FT1_temp/temp[1] <-> Module 1 (IOL_16/4_I/O-Bytes)/TxPDO/input byte 8
//     PlcTask Inputs/Entradas.CA2_L6_FT1_temp/temp[0] <-> Module 3 (IOL_16/4_I/O-Bytes)/TxPDO/input byte 9
//     PlcTask Inputs/Entradas.CA2_L6_FT1_temp/temp[1] <-> Module 3 (IOL_16/4_I/O-Bytes)/TxPDO/input byte 8
//     PlcTask Inputs/Entradas.CA2_L7_FT1_temp/temp[0] <-> Module 5 (IOL_16/4_I/O-Bytes)/TxPDO/input byte 9
//     PlcTask Inputs/Entradas.CA2_L7_FT1_temp/temp[1] <-> Module 5 (IOL_16/4_I/O-Bytes)/TxPDO/input byte 8
//     PlcTask Inputs/Entradas.CA2_L8_FT1_temp/temp[0] <-> Module 7 (IOL_16/4_I/O-Bytes)/TxPDO/input byte 9
//     PlcTask Inputs/Entradas.CA2_L8_FT1_temp/temp[1] <-> Module 7 (IOL_16/4_I/O-Bytes)/TxPDO/input byte 8
//     PlcTask Inputs/Entradas.CA2_L5_FT1_tot/total[0] <-> Module 1 (IOL_16/4_I/O-Bytes)/TxPDO/input byte 3
//     PlcTask Inputs/Entradas.CA2_L5_FT1_tot/total[1] <-> Module 1 (IOL_16/4_I/O-Bytes)/TxPDO/input byte 2
//     PlcTask Inputs/Entradas.CA2_L5_FT1_tot/total[2] <-> Module 1 (IOL_16/4_I/O-Bytes)/TxPDO/input byte 1
//     PlcTask Inputs/Entradas.CA2_L5_FT1_tot/total[3] <-> Module 1 (IOL_16/4_I/O-Bytes)/TxPDO/input byte 0
//     PlcTask Inputs/Entradas.CA2_L6_FT1_tot/total[0] <-> Module 3 (IOL_16/4_I/O-Bytes)/TxPDO/input byte 3
//     PlcTask Inputs/Entradas.CA2_L6_FT1_tot/total[1] <-> Module 3 (IOL_16/4_I/O-Bytes)/TxPDO/input byte 2
//     PlcTask Inputs/Entradas.CA2_L6_FT1_tot/total[2] <-> Module 3 (IOL_16/4_I/O-Bytes)/TxPDO/input byte 1
//     PlcTask Inputs/Entradas.CA2_L6_FT1_tot/total[3] <-> Module 3 (IOL_16/4_I/O-Bytes)/TxPDO/input byte 0
//     PlcTask Inputs/Entradas.CA2_L7_FT1_tot/total[0] <-> Module 5 (IOL_16/4_I/O-Bytes)/TxPDO/input byte 3
//     PlcTask Inputs/Entradas.CA2_L7_FT1_tot/total[1] <-> Module 5 (IOL_16/4_I/O-Bytes)/TxPDO/input byte 2
//     PlcTask Inputs/Entradas.CA2_L7_FT1_tot/total[2] <-> Module 5 (IOL_16/4_I/O-Bytes)/TxPDO/input byte 1
//     PlcTask Inputs/Entradas.CA2_L7_FT1_tot/total[3] <-> Module 5 (IOL_16/4_I/O-Bytes)/TxPDO/input byte 0
//     PlcTask Inputs/Entradas.CA2_L8_FT1_tot/total[0] <-> Module 7 (IOL_16/4_I/O-Bytes)/TxPDO/input byte 3
//     PlcTask Inputs/Entradas.CA2_L8_FT1_tot/total[1] <-> Module 7 (IOL_16/4_I/O-Bytes)/TxPDO/input byte 2
//     PlcTask Inputs/Entradas.CA2_L8_FT1_tot/total[2] <-> Module 7 (IOL_16/4_I/O-Bytes)/TxPDO/input byte 1
//     PlcTask Inputs/Entradas.CA2_L8_FT1_tot/total[3] <-> Module 7 (IOL_16/4_I/O-Bytes)/TxPDO/input byte 0
//     PlcTask Inputs/Entradas.CA2_L5_V1_POSIC/Posicao[0] <-> Module 2 (IOL_4/4_I/O-Bytes)/TxPDO/input byte 0
//     PlcTask Inputs/Entradas.CA2_L5_V1_POSIC/Posicao[1] <-> Module 2 (IOL_4/4_I/O-Bytes)/TxPDO/input byte 1
//     PlcTask Inputs/Entradas.CA2_L6_V1_POSIC/Posicao[0] <-> Module 4 (IOL_4/4_I/O-Bytes)/TxPDO/input byte 0
//     PlcTask Inputs/Entradas.CA2_L6_V1_POSIC/Posicao[1] <-> Module 4 (IOL_4/4_I/O-Bytes)/TxPDO/input byte 1
//     PlcTask Inputs/Entradas.CA2_L7_V1_POSIC/Posicao[0] <-> Module 6 (IOL_4/4_I/O-Bytes)/TxPDO/input byte 0
//     PlcTask Inputs/Entradas.CA2_L7_V1_POSIC/Posicao[1] <-> Module 6 (IOL_4/4_I/O-Bytes)/TxPDO/input byte 1
//     PlcTask Inputs/Entradas.CA2_L8_V1_POSIC/Posicao[0] <-> Module 8 (IOL_4/4_I/O-Bytes)/TxPDO/input byte 0
//     PlcTask Inputs/Entradas.CA2_L8_V1_POSIC/Posicao[1] <-> Module 8 (IOL_4/4_I/O-Bytes)/TxPDO/input byte 1
//     PlcTask Inputs/ioLink.b3St1_CA2_L{5..8}_V1 <-> Module {2..8 step 2} (IOL_4/4_I/O-Bytes)/TxPDO/input byte 3  (4 links)
//     PlcTask Outputs/ioLink.b0Cmd_CA2_L{5..8}_V1 <-> Module {2..8 step 2} (IOL_4/4_I/O-Bytes)/RxPDO/output byte 0  (4 links)
//   Untitled1/Untitled1 Instance <-> Dispositivos (EtherCAT)/C1 (EK1100)/C8 (EK1122)/CA2_2 (EP3356-0022)
//     PlcTask Inputs/Entradas.CA2_WT1_bWcState <-> WcState/WcState
//     PlcTask Inputs/Entradas.CA2_WT1_rValue_REAL <-> RMB Value (Real)/Value (Real)
//     PlcTask Inputs/Entradas.CA2_WT1_stEcSlaveAmsNetAdr <-> InfoData/AdsAddr
//     PlcTask Inputs/Entradas.CA2_WT1_wState <-> RMB Status/Status
//     PlcTask Inputs/Entradas.CA2_WT1_wStatus <-> InfoData/State
//     PlcTask Outputs/Salidas.CA2_WT1_wControl <-> RMB Control/Ctrl
//   Untitled1/Untitled1 Instance <-> Dispositivos (EtherCAT)/C1 (EK1100)/C8 (EK1122)/PU1_1 (EP3356-0022)
//     PlcTask Inputs/Entradas.PU1_WT4_bWcState <-> WcState/WcState
//     PlcTask Inputs/Entradas.PU1_WT4_rValue_REAL <-> RMB Value (Real)/Value (Real)
//     PlcTask Inputs/Entradas.PU1_WT4_stEcSlaveAmsNetAdr <-> InfoData/AdsAddr
//     PlcTask Inputs/Entradas.PU1_WT4_wState <-> InfoData/State
//     PlcTask Inputs/Entradas.PU1_WT4_wStatus <-> RMB Status/Status
//     PlcTask Outputs/Salidas.PU1_WT4_wControl <-> RMB Control/Ctrl
//   Untitled1/Untitled1 Instance <-> Dispositivos (EtherCAT)/C1 (EK1100)/C8 (EK1122)/PU1_2 (ifm IO-Link Master AL1332)
//     PlcTask Inputs/Entradas.CA1_L3_V2_POSIC/Posicao[0] <-> Module 6 (IOL_4/4_I/O-Bytes)/TxPDO/input byte 0
//     PlcTask Inputs/Entradas.CA1_L3_V2_POSIC/Posicao[1] <-> Module 6 (IOL_4/4_I/O-Bytes)/TxPDO/input byte 1
//     PlcTask Inputs/Entradas.CA1_L3_V3_POSIC/Posicao[0] <-> Module 4 (IOL_4/4_I/O-Bytes)/TxPDO/input byte 0
//     PlcTask Inputs/Entradas.CA1_L3_V3_POSIC/Posicao[1] <-> Module 4 (IOL_4/4_I/O-Bytes)/TxPDO/input byte 1
//     PlcTask Inputs/Entradas.CA1_L3_V4_POSIC/Posicao[0] <-> Module 2 (IOL_4/4_I/O-Bytes)/TxPDO/input byte 0
//     PlcTask Inputs/Entradas.CA1_L3_V4_POSIC/Posicao[1] <-> Module 2 (IOL_4/4_I/O-Bytes)/TxPDO/input byte 1
//     PlcTask Inputs/Entradas.CA1_L4_V2_POSIC/Posicao[0] <-> Module 5 (IOL_4/4_I/O-Bytes)/TxPDO/input byte 0
//     PlcTask Inputs/Entradas.CA1_L4_V2_POSIC/Posicao[1] <-> Module 5 (IOL_4/4_I/O-Bytes)/TxPDO/input byte 1
//     PlcTask Inputs/Entradas.CA1_L4_V3_POSIC/Posicao[0] <-> Module 3 (IOL_4/4_I/O-Bytes)/TxPDO/input byte 0
//     PlcTask Inputs/Entradas.CA1_L4_V3_POSIC/Posicao[1] <-> Module 3 (IOL_4/4_I/O-Bytes)/TxPDO/input byte 1
//     PlcTask Inputs/Entradas.CA1_L4_V4_POSIC/Posicao[0] <-> Module 1 (IOL_4/4_I/O-Bytes)/TxPDO/input byte 0
//     PlcTask Inputs/Entradas.CA1_L4_V4_POSIC/Posicao[1] <-> Module 1 (IOL_4/4_I/O-Bytes)/TxPDO/input byte 1
//     PlcTask Inputs/Entradas.bPP1_L3_BD_MangRota <-> Module 8 (Digital_IN)/TxPDO/input byte 0
//     PlcTask Inputs/Entradas.bPP1_L4_BD_MangRota <-> Module 7 (Digital_IN)/TxPDO/input byte 0
//     PlcTask Inputs/ioLink.b3St1_CA1_L3_V2 <-> Module 6 (IOL_4/4_I/O-Bytes)/TxPDO/input byte 3
//     PlcTask Inputs/ioLink.b3St1_CA1_L3_V3 <-> Module 4 (IOL_4/4_I/O-Bytes)/TxPDO/input byte 3
//     PlcTask Inputs/ioLink.b3St1_CA1_L3_V4 <-> Module 2 (IOL_4/4_I/O-Bytes)/TxPDO/input byte 3
//     PlcTask Inputs/ioLink.b3St1_CA1_L4_V2 <-> Module 5 (IOL_4/4_I/O-Bytes)/TxPDO/input byte 3
//     PlcTask Inputs/ioLink.b3St1_CA1_L4_V3 <-> Module 3 (IOL_4/4_I/O-Bytes)/TxPDO/input byte 3
//     PlcTask Inputs/ioLink.b3St1_CA1_L4_V4 <-> Module 1 (IOL_4/4_I/O-Bytes)/TxPDO/input byte 3
//     PlcTask Outputs/ioLink.b0Cmd_CA1_L3_V2 <-> Module 6 (IOL_4/4_I/O-Bytes)/RxPDO/output byte 0
//     PlcTask Outputs/ioLink.b0Cmd_CA1_L3_V3 <-> Module 4 (IOL_4/4_I/O-Bytes)/RxPDO/output byte 0
//     PlcTask Outputs/ioLink.b0Cmd_CA1_L3_V4 <-> Module 2 (IOL_4/4_I/O-Bytes)/RxPDO/output byte 0
//     PlcTask Outputs/ioLink.b0Cmd_CA1_L4_V2 <-> Module 5 (IOL_4/4_I/O-Bytes)/RxPDO/output byte 0
//     PlcTask Outputs/ioLink.b0Cmd_CA1_L4_V3 <-> Module 3 (IOL_4/4_I/O-Bytes)/RxPDO/output byte 0
//     PlcTask Outputs/ioLink.b0Cmd_CA1_L4_V4 <-> Module 1 (IOL_4/4_I/O-Bytes)/RxPDO/output byte 0
//   Untitled1/Untitled1 Instance <-> Dispositivos (EtherCAT)/C1 (EK1100)/C8 (EK1122)/PU1_3 (EP3356-0022)
//     PlcTask Inputs/Entradas.PU1_WT3_bWcState <-> WcState/WcState
//     PlcTask Inputs/Entradas.PU1_WT3_rValue_REAL <-> RMB Value (Real)/Value (Real)
//     PlcTask Inputs/Entradas.PU1_WT3_stEcSlaveAmsNetAdr <-> InfoData/AdsAddr
//     PlcTask Inputs/Entradas.PU1_WT3_wState <-> InfoData/State
//     PlcTask Inputs/Entradas.PU1_WT3_wStatus <-> RMB Status/Status
//     PlcTask Outputs/Salidas.PU1_WT3_wControl <-> RMB Control/Ctrl
//   Untitled1/Untitled1 Instance <-> Dispositivos (EtherCAT)/C1 (EK1100)/C8 (EK1122)/PU1_4 (EP3356-0022)
//     PlcTask Inputs/Entradas.PU1_WT2_bWcState <-> WcState/WcState
//     PlcTask Inputs/Entradas.PU1_WT2_rValue_REAL <-> RMB Value (Real)/Value (Real)
//     PlcTask Inputs/Entradas.PU1_WT2_stEcSlaveAmsNetAdr <-> InfoData/AdsAddr
//     PlcTask Inputs/Entradas.PU1_WT2_wState <-> InfoData/State
//     PlcTask Inputs/Entradas.PU1_WT2_wStatus <-> RMB Status/Status
//     PlcTask Outputs/Salidas.PU1_WT2_wControl <-> RMB Control/Ctrl
//   Untitled1/Untitled1 Instance <-> Dispositivos (EtherCAT)/C1 (EK1100)/C8 (EK1122)/PU1_5 (ifm IO-Link Master AL1332)
//     PlcTask Inputs/Entradas.CA1_L1_V2_POSIC/Posicao[0] <-> Module 5 (IOL_4/4_I/O-Bytes)/TxPDO/input byte 0
//     PlcTask Inputs/Entradas.CA1_L1_V2_POSIC/Posicao[1] <-> Module 5 (IOL_4/4_I/O-Bytes)/TxPDO/input byte 1
//     PlcTask Inputs/Entradas.CA1_L1_V3_POSIC/Posicao[0] <-> Module 3 (IOL_4/4_I/O-Bytes)/TxPDO/input byte 0
//     PlcTask Inputs/Entradas.CA1_L1_V3_POSIC/Posicao[1] <-> Module 3 (IOL_4/4_I/O-Bytes)/TxPDO/input byte 1
//     PlcTask Inputs/Entradas.CA1_L1_V4_POSIC/Posicao[0] <-> Module 1 (IOL_4/4_I/O-Bytes)/TxPDO/input byte 0
//     PlcTask Inputs/Entradas.CA1_L1_V4_POSIC/Posicao[1] <-> Module 1 (IOL_4/4_I/O-Bytes)/TxPDO/input byte 1
//     PlcTask Inputs/Entradas.CA1_L2_V2_POSIC/Posicao[0] <-> Module 6 (IOL_4/4_I/O-Bytes)/TxPDO/input byte 0
//     PlcTask Inputs/Entradas.CA1_L2_V2_POSIC/Posicao[1] <-> Module 6 (IOL_4/4_I/O-Bytes)/TxPDO/input byte 1
//     PlcTask Inputs/Entradas.CA1_L2_V3_POSIC/Posicao[0] <-> Module 4 (IOL_4/4_I/O-Bytes)/TxPDO/input byte 0
//     PlcTask Inputs/Entradas.CA1_L2_V3_POSIC/Posicao[1] <-> Module 4 (IOL_4/4_I/O-Bytes)/TxPDO/input byte 1
//     PlcTask Inputs/Entradas.CA1_L2_V4_POSIC/Posicao[0] <-> Module 2 (IOL_4/4_I/O-Bytes)/TxPDO/input byte 0
//     PlcTask Inputs/Entradas.CA1_L2_V4_POSIC/Posicao[1] <-> Module 2 (IOL_4/4_I/O-Bytes)/TxPDO/input byte 1
//     PlcTask Inputs/Entradas.bPP1_L1_BD_MangRota <-> Module 7 (Digital_IN)/TxPDO/input byte 0
//     PlcTask Inputs/Entradas.bPP1_L2_BD_MangRota <-> Module 8 (Digital_IN)/TxPDO/input byte 0
//     PlcTask Inputs/ioLink.b3St1_CA1_L1_V2 <-> Module 5 (IOL_4/4_I/O-Bytes)/TxPDO/input byte 3
//     PlcTask Inputs/ioLink.b3St1_CA1_L1_V3 <-> Module 3 (IOL_4/4_I/O-Bytes)/TxPDO/input byte 3
//     PlcTask Inputs/ioLink.b3St1_CA1_L1_V4 <-> Module 1 (IOL_4/4_I/O-Bytes)/TxPDO/input byte 3
//     PlcTask Inputs/ioLink.b3St1_CA1_L2_V2 <-> Module 6 (IOL_4/4_I/O-Bytes)/TxPDO/input byte 3
//     PlcTask Inputs/ioLink.b3St1_CA1_L2_V3 <-> Module 4 (IOL_4/4_I/O-Bytes)/TxPDO/input byte 3
//     PlcTask Inputs/ioLink.b3St1_CA1_L2_V4 <-> Module 2 (IOL_4/4_I/O-Bytes)/TxPDO/input byte 3
//     PlcTask Outputs/ioLink.b0Cmd_CA1_L1_V2 <-> Module 5 (IOL_4/4_I/O-Bytes)/RxPDO/output byte 0
//     PlcTask Outputs/ioLink.b0Cmd_CA1_L1_V3 <-> Module 3 (IOL_4/4_I/O-Bytes)/RxPDO/output byte 0
//     PlcTask Outputs/ioLink.b0Cmd_CA1_L1_V4 <-> Module 1 (IOL_4/4_I/O-Bytes)/RxPDO/output byte 0
//     PlcTask Outputs/ioLink.b0Cmd_CA1_L2_V2 <-> Module 6 (IOL_4/4_I/O-Bytes)/RxPDO/output byte 0
//     PlcTask Outputs/ioLink.b0Cmd_CA1_L2_V3 <-> Module 4 (IOL_4/4_I/O-Bytes)/RxPDO/output byte 0
//     PlcTask Outputs/ioLink.b0Cmd_CA1_L2_V4 <-> Module 2 (IOL_4/4_I/O-Bytes)/RxPDO/output byte 0
//   Untitled1/Untitled1 Instance <-> Dispositivos (EtherCAT)/C1 (EK1100)/C8 (EK1122)/PU1_6 (EP3356-0022)
//     PlcTask Inputs/Entradas.PU1_WT1_bWcState <-> WcState/WcState
//     PlcTask Inputs/Entradas.PU1_WT1_rValue_REAL <-> RMB Value (Real)/Value (Real)
//     PlcTask Inputs/Entradas.PU1_WT1_stEcSlaveAmsNetAdr <-> InfoData/AdsAddr
//     PlcTask Inputs/Entradas.PU1_WT1_wState <-> RMB Status/Status
//     PlcTask Inputs/Entradas.PU1_WT1_wStatus <-> InfoData/State
//     PlcTask Outputs/Salidas.PU1_WT1_wControl <-> RMB Control/Ctrl
//   Untitled1/Untitled1 Instance <-> Dispositivos (EtherCAT)/C1 (EK1100)/C8 (EK1122)/PU2_1 (EP3356-0022)
//     PlcTask Inputs/Entradas.PU2_WT8_bWcState <-> WcState/WcState
//     PlcTask Inputs/Entradas.PU2_WT8_rValue_REAL <-> RMB Value (Real)/Value (Real)
//     PlcTask Inputs/Entradas.PU2_WT8_stEcSlaveAmsNetAdr <-> InfoData/AdsAddr
//     PlcTask Inputs/Entradas.PU2_WT8_wState <-> RMB Status/Status
//     PlcTask Inputs/Entradas.PU2_WT8_wStatus <-> InfoData/State
//     PlcTask Outputs/Salidas.PU2_WT8_wControl <-> RMB Control/Ctrl
//   Untitled1/Untitled1 Instance <-> Dispositivos (EtherCAT)/C1 (EK1100)/C8 (EK1122)/PU2_2 (ifm IO-Link Master AL1332)
//     PlcTask Inputs/Entradas.CA2_L7_V2_POSIC/Posicao[0] <-> Module 6 (IOL_4/4_I/O-Bytes)/TxPDO/input byte 0
//     PlcTask Inputs/Entradas.CA2_L7_V2_POSIC/Posicao[1] <-> Module 6 (IOL_4/4_I/O-Bytes)/TxPDO/input byte 1
//     PlcTask Inputs/Entradas.CA2_L7_V3_POSIC/Posicao[0] <-> Module 4 (IOL_4/4_I/O-Bytes)/TxPDO/input byte 0
//     PlcTask Inputs/Entradas.CA2_L7_V3_POSIC/Posicao[1] <-> Module 4 (IOL_4/4_I/O-Bytes)/TxPDO/input byte 1
//     PlcTask Inputs/Entradas.CA2_L7_V4_POSIC/Posicao[0] <-> Module 2 (IOL_4/4_I/O-Bytes)/TxPDO/input byte 0
//     PlcTask Inputs/Entradas.CA2_L7_V4_POSIC/Posicao[1] <-> Module 2 (IOL_4/4_I/O-Bytes)/TxPDO/input byte 1
//     PlcTask Inputs/Entradas.CA2_L8_V2_POSIC/Posicao[0] <-> Module 5 (IOL_4/4_I/O-Bytes)/TxPDO/input byte 0
//     PlcTask Inputs/Entradas.CA2_L8_V2_POSIC/Posicao[1] <-> Module 5 (IOL_4/4_I/O-Bytes)/TxPDO/input byte 1
//     PlcTask Inputs/Entradas.CA2_L8_V3_POSIC/Posicao[0] <-> Module 3 (IOL_4/4_I/O-Bytes)/TxPDO/input byte 0
//     PlcTask Inputs/Entradas.CA2_L8_V3_POSIC/Posicao[1] <-> Module 3 (IOL_4/4_I/O-Bytes)/TxPDO/input byte 1
//     PlcTask Inputs/Entradas.CA2_L8_V4_POSIC/Posicao[0] <-> Module 1 (IOL_4/4_I/O-Bytes)/TxPDO/input byte 0
//     PlcTask Inputs/Entradas.CA2_L8_V4_POSIC/Posicao[1] <-> Module 1 (IOL_4/4_I/O-Bytes)/TxPDO/input byte 1
//     PlcTask Inputs/Entradas.bPP2_L7_BD_MangRota <-> Module 8 (Digital_IN)/TxPDO/input byte 0
//     PlcTask Inputs/Entradas.bPP2_L8_BD_MangRota <-> Module 7 (Digital_IN)/TxPDO/input byte 0
//     PlcTask Inputs/ioLink.b3St1_CA2_L7_V2 <-> Module 6 (IOL_4/4_I/O-Bytes)/TxPDO/input byte 3
//     PlcTask Inputs/ioLink.b3St1_CA2_L7_V3 <-> Module 4 (IOL_4/4_I/O-Bytes)/TxPDO/input byte 3
//     PlcTask Inputs/ioLink.b3St1_CA2_L7_V4 <-> Module 2 (IOL_4/4_I/O-Bytes)/TxPDO/input byte 3
//     PlcTask Inputs/ioLink.b3St1_CA2_L8_V2 <-> Module 5 (IOL_4/4_I/O-Bytes)/TxPDO/input byte 3
//     PlcTask Inputs/ioLink.b3St1_CA2_L8_V3 <-> Module 3 (IOL_4/4_I/O-Bytes)/TxPDO/input byte 3
//     PlcTask Inputs/ioLink.b3St1_CA2_L8_V4 <-> Module 1 (IOL_4/4_I/O-Bytes)/TxPDO/input byte 3
//     PlcTask Outputs/ioLink.b0Cmd_CA2_L7_V2 <-> Module 6 (IOL_4/4_I/O-Bytes)/RxPDO/output byte 0
//     PlcTask Outputs/ioLink.b0Cmd_CA2_L7_V3 <-> Module 4 (IOL_4/4_I/O-Bytes)/RxPDO/output byte 0
//     PlcTask Outputs/ioLink.b0Cmd_CA2_L7_V4 <-> Module 2 (IOL_4/4_I/O-Bytes)/RxPDO/output byte 0
//     PlcTask Outputs/ioLink.b0Cmd_CA2_L8_V2 <-> Module 5 (IOL_4/4_I/O-Bytes)/RxPDO/output byte 0
//     PlcTask Outputs/ioLink.b0Cmd_CA2_L8_V3 <-> Module 3 (IOL_4/4_I/O-Bytes)/RxPDO/output byte 0
//     PlcTask Outputs/ioLink.b0Cmd_CA2_L8_V4 <-> Module 1 (IOL_4/4_I/O-Bytes)/RxPDO/output byte 0
//   Untitled1/Untitled1 Instance <-> Dispositivos (EtherCAT)/C1 (EK1100)/C8 (EK1122)/PU2_3 (EP3356-0022)
//     PlcTask Inputs/Entradas.PU2_WT7_bWcState <-> WcState/WcState
//     PlcTask Inputs/Entradas.PU2_WT7_rValue_REAL <-> RMB Value (Real)/Value (Real)
//     PlcTask Inputs/Entradas.PU2_WT7_stEcSlaveAmsNetAdr <-> InfoData/AdsAddr
//     PlcTask Inputs/Entradas.PU2_WT7_wState <-> InfoData/State
//     PlcTask Inputs/Entradas.PU2_WT7_wStatus <-> RMB Status/Status
//     PlcTask Outputs/Salidas.PU2_WT7_wControl <-> RMB Control/Ctrl
//   Untitled1/Untitled1 Instance <-> Dispositivos (EtherCAT)/C1 (EK1100)/C8 (EK1122)/PU2_4 (EP3356-0022)
//     PlcTask Inputs/Entradas.PU2_WT6_bWcState <-> WcState/WcState
//     PlcTask Inputs/Entradas.PU2_WT6_rValue_REAL <-> RMB Value (Real)/Value (Real)
//     PlcTask Inputs/Entradas.PU2_WT6_stEcSlaveAmsNetAdr <-> InfoData/AdsAddr
//     PlcTask Inputs/Entradas.PU2_WT6_wState <-> InfoData/State
//     PlcTask Inputs/Entradas.PU2_WT6_wStatus <-> RMB Status/Status
//     PlcTask Outputs/Salidas.PU2_WT6_wControl <-> RMB Control/Ctrl
//   Untitled1/Untitled1 Instance <-> Dispositivos (EtherCAT)/C1 (EK1100)/C8 (EK1122)/PU2_5 (ifm IO-Link Master AL1332)
//     PlcTask Inputs/Entradas.CA2_L5_V2_POSIC/Posicao[0] <-> Module 5 (IOL_4/4_I/O-Bytes)/TxPDO/input byte 0
//     PlcTask Inputs/Entradas.CA2_L5_V2_POSIC/Posicao[1] <-> Module 5 (IOL_4/4_I/O-Bytes)/TxPDO/input byte 1
//     PlcTask Inputs/Entradas.CA2_L5_V3_POSIC/Posicao[0] <-> Module 3 (IOL_4/4_I/O-Bytes)/TxPDO/input byte 0
//     PlcTask Inputs/Entradas.CA2_L5_V3_POSIC/Posicao[1] <-> Module 3 (IOL_4/4_I/O-Bytes)/TxPDO/input byte 1
//     PlcTask Inputs/Entradas.CA2_L5_V4_POSIC/Posicao[0] <-> Module 1 (IOL_4/4_I/O-Bytes)/TxPDO/input byte 0
//     PlcTask Inputs/Entradas.CA2_L5_V4_POSIC/Posicao[1] <-> Module 1 (IOL_4/4_I/O-Bytes)/TxPDO/input byte 1
//     PlcTask Inputs/Entradas.CA2_L6_V2_POSIC/Posicao[0] <-> Module 6 (IOL_4/4_I/O-Bytes)/TxPDO/input byte 0
//     PlcTask Inputs/Entradas.CA2_L6_V2_POSIC/Posicao[1] <-> Module 6 (IOL_4/4_I/O-Bytes)/TxPDO/input byte 1
//     PlcTask Inputs/Entradas.CA2_L6_V3_POSIC/Posicao[0] <-> Module 4 (IOL_4/4_I/O-Bytes)/TxPDO/input byte 0
//     PlcTask Inputs/Entradas.CA2_L6_V3_POSIC/Posicao[1] <-> Module 4 (IOL_4/4_I/O-Bytes)/TxPDO/input byte 1
//     PlcTask Inputs/Entradas.CA2_L6_V4_POSIC/Posicao[0] <-> Module 2 (IOL_4/4_I/O-Bytes)/TxPDO/input byte 0
//     PlcTask Inputs/Entradas.CA2_L6_V4_POSIC/Posicao[1] <-> Module 2 (IOL_4/4_I/O-Bytes)/TxPDO/input byte 1
//     PlcTask Inputs/Entradas.bPP2_L5_BD_MangRota <-> Module 7 (Digital_IN)/TxPDO/input byte 0
//     PlcTask Inputs/Entradas.bPP2_L6_BD_MangRota <-> Module 8 (Digital_IN)/TxPDO/input byte 0
//     PlcTask Inputs/ioLink.b3St1_CA2_L5_V2 <-> Module 5 (IOL_4/4_I/O-Bytes)/TxPDO/input byte 3
//     PlcTask Inputs/ioLink.b3St1_CA2_L5_V3 <-> Module 3 (IOL_4/4_I/O-Bytes)/TxPDO/input byte 3
//     PlcTask Inputs/ioLink.b3St1_CA2_L5_V4 <-> Module 1 (IOL_4/4_I/O-Bytes)/TxPDO/input byte 3
//     PlcTask Inputs/ioLink.b3St1_CA2_L6_V2 <-> Module 6 (IOL_4/4_I/O-Bytes)/TxPDO/input byte 3
//     PlcTask Inputs/ioLink.b3St1_CA2_L6_V3 <-> Module 4 (IOL_4/4_I/O-Bytes)/TxPDO/input byte 3
//     PlcTask Inputs/ioLink.b3St1_CA2_L6_V4 <-> Module 2 (IOL_4/4_I/O-Bytes)/TxPDO/input byte 3
//     PlcTask Outputs/ioLink.b0Cmd_CA2_L5_V2 <-> Module 5 (IOL_4/4_I/O-Bytes)/RxPDO/output byte 0
//     PlcTask Outputs/ioLink.b0Cmd_CA2_L5_V3 <-> Module 3 (IOL_4/4_I/O-Bytes)/RxPDO/output byte 0
//     PlcTask Outputs/ioLink.b0Cmd_CA2_L5_V4 <-> Module 1 (IOL_4/4_I/O-Bytes)/RxPDO/output byte 0
//     PlcTask Outputs/ioLink.b0Cmd_CA2_L6_V2 <-> Module 6 (IOL_4/4_I/O-Bytes)/RxPDO/output byte 0
//     PlcTask Outputs/ioLink.b0Cmd_CA2_L6_V3 <-> Module 4 (IOL_4/4_I/O-Bytes)/RxPDO/output byte 0
//     PlcTask Outputs/ioLink.b0Cmd_CA2_L6_V4 <-> Module 2 (IOL_4/4_I/O-Bytes)/RxPDO/output byte 0
//   Untitled1/Untitled1 Instance <-> Dispositivos (EtherCAT)/C1 (EK1100)/C8 (EK1122)/PU2_6 (EP3356-0022)
//     PlcTask Inputs/Entradas.PU2_WT5_bWcState <-> WcState/WcState
//     PlcTask Inputs/Entradas.PU2_WT5_rValue_REAL <-> RMB Value (Real)/Value (Real)
//     PlcTask Inputs/Entradas.PU2_WT5_stEcSlaveAmsNetAdr <-> InfoData/AdsAddr
//     PlcTask Inputs/Entradas.PU2_WT5_wState <-> InfoData/State
//     PlcTask Inputs/Entradas.PU2_WT5_wStatus <-> RMB Status/Status
//     PlcTask Outputs/Salidas.PU2_WT5_wControl <-> RMB Control/Ctrl
//   Untitled1/Untitled1 Instance <-> Dispositivos (EtherCAT)/C1 (EK1100)/C8 (EK1122)/PU4_1 (ifm IO-Link Master AL1330)
//     PlcTask Inputs/ioLink.b3St1_PU_Lav_V5 <-> Module 2 (IOL_4/4_I/O-Bytes)/TxPDO/input byte 3
//     PlcTask Inputs/ioLink.b3St1_PU_Lav_V6 <-> Module 1 (IOL_4/4_I/O-Bytes)/TxPDO/input byte 3
//     PlcTask Outputs/ioLink.b0Cmd_PU_Lav_V5 <-> Module 2 (IOL_4/4_I/O-Bytes)/RxPDO/output byte 0
//     PlcTask Outputs/ioLink.b0Cmd_PU_Lav_V6 <-> Module 1 (IOL_4/4_I/O-Bytes)/RxPDO/output byte 0
//   Untitled1/Untitled1 Instance <-> Dispositivos (EtherCAT)/C1 (EK1100)/C9 (EK1122)/CA3_1 (ifm IO-Link Master AL1332)
//     PlcTask Inputs/Entradas.CA3_L10_FT1_caudal/caudal[0] <-> Module 3 (IOL_16/4_I/O-Bytes)/TxPDO/input byte 5
//     PlcTask Inputs/Entradas.CA3_L10_FT1_caudal/caudal[1] <-> Module 3 (IOL_16/4_I/O-Bytes)/TxPDO/input byte 4
//     PlcTask Inputs/Entradas.CA3_L11_FT1_caudal/caudal[0] <-> Module 5 (IOL_16/4_I/O-Bytes)/TxPDO/input byte 5
//     PlcTask Inputs/Entradas.CA3_L11_FT1_caudal/caudal[1] <-> Module 5 (IOL_16/4_I/O-Bytes)/TxPDO/input byte 4
//     PlcTask Inputs/Entradas.CA3_L12_FT1_caudal/caudal[0] <-> Module 7 (IOL_16/4_I/O-Bytes)/TxPDO/input byte 5
//     PlcTask Inputs/Entradas.CA3_L12_FT1_caudal/caudal[1] <-> Module 7 (IOL_16/4_I/O-Bytes)/TxPDO/input byte 4
//     PlcTask Inputs/Entradas.CA3_L9_FT1_caudal/caudal[0] <-> Module 1 (IOL_16/4_I/O-Bytes)/TxPDO/input byte 5
//     PlcTask Inputs/Entradas.CA3_L9_FT1_caudal/caudal[1] <-> Module 1 (IOL_16/4_I/O-Bytes)/TxPDO/input byte 4
//     PlcTask Inputs/Entradas.CA3_L10_FT1_temp/temp[0] <-> Module 3 (IOL_16/4_I/O-Bytes)/TxPDO/input byte 9
//     PlcTask Inputs/Entradas.CA3_L10_FT1_temp/temp[1] <-> Module 3 (IOL_16/4_I/O-Bytes)/TxPDO/input byte 8
//     PlcTask Inputs/Entradas.CA3_L11_FT1_temp/temp[0] <-> Module 5 (IOL_16/4_I/O-Bytes)/TxPDO/input byte 9
//     PlcTask Inputs/Entradas.CA3_L11_FT1_temp/temp[1] <-> Module 5 (IOL_16/4_I/O-Bytes)/TxPDO/input byte 8
//     PlcTask Inputs/Entradas.CA3_L12_FT1_temp/temp[0] <-> Module 7 (IOL_16/4_I/O-Bytes)/TxPDO/input byte 9
//     PlcTask Inputs/Entradas.CA3_L12_FT1_temp/temp[1] <-> Module 7 (IOL_16/4_I/O-Bytes)/TxPDO/input byte 8
//     PlcTask Inputs/Entradas.CA3_L9_FT1_temp/temp[0] <-> Module 1 (IOL_16/4_I/O-Bytes)/TxPDO/input byte 9
//     PlcTask Inputs/Entradas.CA3_L9_FT1_temp/temp[1] <-> Module 1 (IOL_16/4_I/O-Bytes)/TxPDO/input byte 8
//     PlcTask Inputs/Entradas.CA3_L10_FT1_tot/total[0] <-> Module 3 (IOL_16/4_I/O-Bytes)/TxPDO/input byte 3
//     PlcTask Inputs/Entradas.CA3_L10_FT1_tot/total[1] <-> Module 3 (IOL_16/4_I/O-Bytes)/TxPDO/input byte 2
//     PlcTask Inputs/Entradas.CA3_L10_FT1_tot/total[2] <-> Module 3 (IOL_16/4_I/O-Bytes)/TxPDO/input byte 1
//     PlcTask Inputs/Entradas.CA3_L10_FT1_tot/total[3] <-> Module 3 (IOL_16/4_I/O-Bytes)/TxPDO/input byte 0
//     PlcTask Inputs/Entradas.CA3_L11_FT1_tot/total[0] <-> Module 5 (IOL_16/4_I/O-Bytes)/TxPDO/input byte 3
//     PlcTask Inputs/Entradas.CA3_L11_FT1_tot/total[1] <-> Module 5 (IOL_16/4_I/O-Bytes)/TxPDO/input byte 2
//     PlcTask Inputs/Entradas.CA3_L11_FT1_tot/total[2] <-> Module 5 (IOL_16/4_I/O-Bytes)/TxPDO/input byte 1
//     PlcTask Inputs/Entradas.CA3_L11_FT1_tot/total[3] <-> Module 5 (IOL_16/4_I/O-Bytes)/TxPDO/input byte 0
//     PlcTask Inputs/Entradas.CA3_L12_FT1_tot/total[0] <-> Module 7 (IOL_16/4_I/O-Bytes)/TxPDO/input byte 3
//     PlcTask Inputs/Entradas.CA3_L12_FT1_tot/total[1] <-> Module 7 (IOL_16/4_I/O-Bytes)/TxPDO/input byte 2
//     PlcTask Inputs/Entradas.CA3_L12_FT1_tot/total[2] <-> Module 7 (IOL_16/4_I/O-Bytes)/TxPDO/input byte 1
//     PlcTask Inputs/Entradas.CA3_L12_FT1_tot/total[3] <-> Module 7 (IOL_16/4_I/O-Bytes)/TxPDO/input byte 0
//     PlcTask Inputs/Entradas.CA3_L9_FT1_tot/total[0] <-> Module 1 (IOL_16/4_I/O-Bytes)/TxPDO/input byte 3
//     PlcTask Inputs/Entradas.CA3_L9_FT1_tot/total[1] <-> Module 1 (IOL_16/4_I/O-Bytes)/TxPDO/input byte 2
//     PlcTask Inputs/Entradas.CA3_L9_FT1_tot/total[2] <-> Module 1 (IOL_16/4_I/O-Bytes)/TxPDO/input byte 1
//     PlcTask Inputs/Entradas.CA3_L9_FT1_tot/total[3] <-> Module 1 (IOL_16/4_I/O-Bytes)/TxPDO/input byte 0
//     PlcTask Inputs/Entradas.CA3_L10_V1_POSIC/Posicao[0] <-> Module 4 (IOL_4/4_I/O-Bytes)/TxPDO/input byte 0
//     PlcTask Inputs/Entradas.CA3_L10_V1_POSIC/Posicao[1] <-> Module 4 (IOL_4/4_I/O-Bytes)/TxPDO/input byte 1
//     PlcTask Inputs/Entradas.CA3_L11_V1_POSIC/Posicao[0] <-> Module 6 (IOL_4/4_I/O-Bytes)/TxPDO/input byte 0
//     PlcTask Inputs/Entradas.CA3_L11_V1_POSIC/Posicao[1] <-> Module 6 (IOL_4/4_I/O-Bytes)/TxPDO/input byte 1
//     PlcTask Inputs/Entradas.CA3_L12_V1_POSIC/Posicao[0] <-> Module 8 (IOL_4/4_I/O-Bytes)/TxPDO/input byte 0
//     PlcTask Inputs/Entradas.CA3_L12_V1_POSIC/Posicao[1] <-> Module 8 (IOL_4/4_I/O-Bytes)/TxPDO/input byte 1
//     PlcTask Inputs/Entradas.CA3_L9_V1_POSIC/Posicao[0] <-> Module 2 (IOL_4/4_I/O-Bytes)/TxPDO/input byte 0
//     PlcTask Inputs/Entradas.CA3_L9_V1_POSIC/Posicao[1] <-> Module 2 (IOL_4/4_I/O-Bytes)/TxPDO/input byte 1
//     PlcTask Inputs/ioLink.b3St1_CA3_L{9..12}_V1 <-> Module {2..8 step 2} (IOL_4/4_I/O-Bytes)/TxPDO/input byte 3  (4 links)
//     PlcTask Outputs/ioLink.b0Cmd_CA3_L{9..12}_V1 <-> Module {2..8 step 2} (IOL_4/4_I/O-Bytes)/RxPDO/output byte 0  (4 links)
//   Untitled1/Untitled1 Instance <-> Dispositivos (EtherCAT)/C1 (EK1100)/C9 (EK1122)/CA3_2 (EP3356-0022)
//     PlcTask Inputs/Entradas.CA3_WT1_bWcState <-> WcState/WcState
//     PlcTask Inputs/Entradas.CA3_WT1_rValue_REAL <-> RMB Value (Real)/Value (Real)
//     PlcTask Inputs/Entradas.CA3_WT1_stEcSlaveAmsNetAdr <-> InfoData/AdsAddr
//     PlcTask Inputs/Entradas.CA3_WT1_wState <-> InfoData/State
//     PlcTask Inputs/Entradas.CA3_WT1_wStatus <-> RMB Status/Status
//     PlcTask Outputs/Salidas.CA3_WT1_wControl <-> RMB Control/Ctrl
//   Untitled1/Untitled1 Instance <-> Dispositivos (EtherCAT)/C1 (EK1100)/C9 (EK1122)/PE_1 (EX260-SEC1)
//     PlcTask Outputs/Salidas.PE_B1_V2 <-> Byte 0/Output[0]
//     PlcTask Outputs/Salidas.PE_B2_V2 <-> Byte 0/Output[2]
//     PlcTask Outputs/Salidas.PE_B3_V2 <-> Byte 0/Output[4]
//     PlcTask Outputs/Salidas.PE_B3_V3 <-> Byte 0/Output[6]
//   Untitled1/Untitled1 Instance <-> Dispositivos (EtherCAT)/C1 (EK1100)/C9 (EK1122)/PE_2 (ifm IO-Link Master AL1332)
//     PlcTask Inputs/Entradas.PE_B1_HLS <-> Module 2 (IOL_4/4_I/O-Bytes)/TxPDO/input byte 1
//     PlcTask Inputs/Entradas.PE_B2_HLS <-> Module 3 (IOL_4/4_I/O-Bytes)/TxPDO/input byte 1
//     PlcTask Inputs/Entradas.PE_B3_HLS <-> Module 4 (IOL_4/4_I/O-Bytes)/TxPDO/input byte 1
//     PlcTask Inputs/Entradas.PE_B1_LLS <-> Module 5 (IOL_4/4_I/O-Bytes)/TxPDO/input byte 1
//     PlcTask Inputs/Entradas.PE_B2_LLS <-> Module 6 (IOL_4/4_I/O-Bytes)/TxPDO/input byte 1
//     PlcTask Inputs/Entradas.PE_B3_LLS <-> Module 7 (IOL_4/4_I/O-Bytes)/TxPDO/input byte 1
//     PlcTask Inputs/Entradas.PE_H_HLS <-> Module 1 (IOL_4/4_I/O-Bytes)/TxPDO/input byte 1
//   Untitled1/Untitled1 Instance <-> Dispositivos (EtherCAT)/C1 (EK1100)/C9 (EK1122)/PE_3 (EX260-SEC1)
//     PlcTask Outputs/Salidas.PE_B1_V1_Pos1 <-> Byte 0/Output[0]
//     PlcTask Outputs/Salidas.PE_B1_V1_Pos2 <-> Byte 0/Output[1]
//     PlcTask Outputs/Salidas.PE_B2_V1_Pos1 <-> Byte 0/Output[2]
//     PlcTask Outputs/Salidas.PE_B2_V1_Pos2 <-> Byte 0/Output[3]
//     PlcTask Outputs/Salidas.PE_B3_V1_Pos1 <-> Byte 0/Output[4]
//     PlcTask Outputs/Salidas.PE_B3_V1_Pos2 <-> Byte 0/Output[5]
//   Untitled1/Untitled1 Instance <-> Dispositivos (EtherCAT)/C1 (EK1100)/C9 (EK1122)/PE_4 (ifm IO-Link Master AL1330)
//     PlcTask Inputs/Entradas.PE_B1_V1_ZO <-> Module 2 (Digital_IN)/TxPDO/input byte 0
//     PlcTask Inputs/Entradas.PE_B2_V1_ZO <-> Module 4 (Digital_IN)/TxPDO/input byte 0
//     PlcTask Inputs/Entradas.PE_B3_V1_ZO <-> Module 3 (Digital_IN)/TxPDO/input byte 0
//     PlcTask Inputs/Entradas.TR_CDT_LLS <-> Module 1 (IOL_4/4_I/O-Bytes)/TxPDO/input byte 1
//   Untitled1/Untitled1 Instance <-> Dispositivos (EtherCAT)/C1 (EK1100)/C9 (EK1122)/PU3_1 (EP3356-0022)
//     PlcTask Inputs/Entradas.PU3_WT12_bWcState <-> WcState/WcState
//     PlcTask Inputs/Entradas.PU3_WT12_rValue_REAL <-> RMB Value (Real)/Value (Real)
//     PlcTask Inputs/Entradas.PU3_WT12_stEcSlaveAmsNetAdr <-> InfoData/AdsAddr
//     PlcTask Inputs/Entradas.PU3_WT12_wState <-> InfoData/State
//     PlcTask Inputs/Entradas.PU3_WT12_wStatus <-> RMB Status/Status
//     PlcTask Outputs/Salidas.PU3_WT12_wControl <-> RMB Control/Ctrl
//   Untitled1/Untitled1 Instance <-> Dispositivos (EtherCAT)/C1 (EK1100)/C9 (EK1122)/PU3_2 (ifm IO-Link Master AL1332)
//     PlcTask Inputs/Entradas.CA3_L11_V2_POSIC/Posicao[0] <-> Module 6 (IOL_4/4_I/O-Bytes)/TxPDO/input byte 0
//     PlcTask Inputs/Entradas.CA3_L11_V2_POSIC/Posicao[1] <-> Module 6 (IOL_4/4_I/O-Bytes)/TxPDO/input byte 1
//     PlcTask Inputs/Entradas.CA3_L11_V3_POSIC/Posicao[0] <-> Module 4 (IOL_4/4_I/O-Bytes)/TxPDO/input byte 0
//     PlcTask Inputs/Entradas.CA3_L11_V3_POSIC/Posicao[1] <-> Module 4 (IOL_4/4_I/O-Bytes)/TxPDO/input byte 1
//     PlcTask Inputs/Entradas.CA3_L11_V4_POSIC/Posicao[0] <-> Module 2 (IOL_4/4_I/O-Bytes)/TxPDO/input byte 0
//     PlcTask Inputs/Entradas.CA3_L11_V4_POSIC/Posicao[1] <-> Module 2 (IOL_4/4_I/O-Bytes)/TxPDO/input byte 1
//     PlcTask Inputs/Entradas.CA3_L12_V2_POSIC/Posicao[0] <-> Module 5 (IOL_4/4_I/O-Bytes)/TxPDO/input byte 0
//     PlcTask Inputs/Entradas.CA3_L12_V2_POSIC/Posicao[1] <-> Module 5 (IOL_4/4_I/O-Bytes)/TxPDO/input byte 1
//     PlcTask Inputs/Entradas.CA3_L12_V3_POSIC/Posicao[0] <-> Module 3 (IOL_4/4_I/O-Bytes)/TxPDO/input byte 0
//     PlcTask Inputs/Entradas.CA3_L12_V3_POSIC/Posicao[1] <-> Module 3 (IOL_4/4_I/O-Bytes)/TxPDO/input byte 1
//     PlcTask Inputs/Entradas.CA3_L12_V4_POSIC/Posicao[0] <-> Module 1 (IOL_4/4_I/O-Bytes)/TxPDO/input byte 0
//     PlcTask Inputs/Entradas.CA3_L12_V4_POSIC/Posicao[1] <-> Module 1 (IOL_4/4_I/O-Bytes)/TxPDO/input byte 1
//     PlcTask Inputs/Entradas.bPP3_L11_BD_MangRota <-> Module 8 (Digital_IN)/TxPDO/input byte 0
//     PlcTask Inputs/Entradas.bPP3_L12_BD_MangRota <-> Module 7 (Digital_IN)/TxPDO/input byte 0
//     PlcTask Inputs/ioLink.b3St1_CA3_L11_V2 <-> Module 6 (IOL_4/4_I/O-Bytes)/TxPDO/input byte 3
//     PlcTask Inputs/ioLink.b3St1_CA3_L11_V3 <-> Module 4 (IOL_4/4_I/O-Bytes)/TxPDO/input byte 3
//     PlcTask Inputs/ioLink.b3St1_CA3_L11_V4 <-> Module 2 (IOL_4/4_I/O-Bytes)/TxPDO/input byte 3
//     PlcTask Inputs/ioLink.b3St1_CA3_L12_V2 <-> Module 5 (IOL_4/4_I/O-Bytes)/TxPDO/input byte 3
//     PlcTask Inputs/ioLink.b3St1_CA3_L12_V3 <-> Module 3 (IOL_4/4_I/O-Bytes)/TxPDO/input byte 3
//     PlcTask Inputs/ioLink.b3St1_CA3_L12_V4 <-> Module 1 (IOL_4/4_I/O-Bytes)/TxPDO/input byte 3
//     PlcTask Outputs/ioLink.b0Cmd_CA3_L11_V2 <-> Module 6 (IOL_4/4_I/O-Bytes)/RxPDO/output byte 0
//     PlcTask Outputs/ioLink.b0Cmd_CA3_L11_V3 <-> Module 4 (IOL_4/4_I/O-Bytes)/RxPDO/output byte 0
//     PlcTask Outputs/ioLink.b0Cmd_CA3_L11_V4 <-> Module 2 (IOL_4/4_I/O-Bytes)/RxPDO/output byte 0
//     PlcTask Outputs/ioLink.b0Cmd_CA3_L12_V2 <-> Module 5 (IOL_4/4_I/O-Bytes)/RxPDO/output byte 0
//     PlcTask Outputs/ioLink.b0Cmd_CA3_L12_V3 <-> Module 3 (IOL_4/4_I/O-Bytes)/RxPDO/output byte 0
//     PlcTask Outputs/ioLink.b0Cmd_CA3_L12_V4 <-> Module 1 (IOL_4/4_I/O-Bytes)/RxPDO/output byte 0
//   Untitled1/Untitled1 Instance <-> Dispositivos (EtherCAT)/C1 (EK1100)/C9 (EK1122)/PU3_3 (EP3356-0022)
//     PlcTask Inputs/Entradas.PU3_WT11_bWcState <-> WcState/WcState
//     PlcTask Inputs/Entradas.PU3_WT11_rValue_REAL <-> RMB Value (Real)/Value (Real)
//     PlcTask Inputs/Entradas.PU3_WT11_stEcSlaveAmsNetAdr <-> InfoData/AdsAddr
//     PlcTask Inputs/Entradas.PU3_WT11_wState <-> InfoData/State
//     PlcTask Inputs/Entradas.PU3_WT11_wStatus <-> RMB Status/Status
//     PlcTask Outputs/Salidas.PU3_WT11_wControl <-> RMB Control/Ctrl
//   Untitled1/Untitled1 Instance <-> Dispositivos (EtherCAT)/C1 (EK1100)/C9 (EK1122)/PU3_4 (EP3356-0022)
//     PlcTask Inputs/Entradas.PU3_WT10_bWcState <-> WcState/WcState
//     PlcTask Inputs/Entradas.PU3_WT10_rValue_REAL <-> RMB Value (Real)/Value (Real)
//     PlcTask Inputs/Entradas.PU3_WT10_stEcSlaveAmsNetAdr <-> InfoData/AdsAddr
//     PlcTask Inputs/Entradas.PU3_WT10_wState <-> InfoData/State
//     PlcTask Inputs/Entradas.PU3_WT10_wStatus <-> RMB Status/Status
//     PlcTask Outputs/Salidas.PU3_WT10_wControl <-> RMB Control/Ctrl
//   Untitled1/Untitled1 Instance <-> Dispositivos (EtherCAT)/C1 (EK1100)/C9 (EK1122)/PU3_5 (ifm IO-Link Master AL1332)
//     PlcTask Inputs/Entradas.CA3_L10_V2_POSIC/Posicao[0] <-> Module 5 (IOL_4/4_I/O-Bytes)/TxPDO/input byte 0
//     PlcTask Inputs/Entradas.CA3_L10_V2_POSIC/Posicao[1] <-> Module 5 (IOL_4/4_I/O-Bytes)/TxPDO/input byte 1
//     PlcTask Inputs/Entradas.CA3_L10_V3_POSIC/Posicao[0] <-> Module 3 (IOL_4/4_I/O-Bytes)/TxPDO/input byte 0
//     PlcTask Inputs/Entradas.CA3_L10_V3_POSIC/Posicao[1] <-> Module 3 (IOL_4/4_I/O-Bytes)/TxPDO/input byte 1
//     PlcTask Inputs/Entradas.CA3_L10_V4_POSIC/Posicao[0] <-> Module 1 (IOL_4/4_I/O-Bytes)/TxPDO/input byte 0
//     PlcTask Inputs/Entradas.CA3_L10_V4_POSIC/Posicao[1] <-> Module 1 (IOL_4/4_I/O-Bytes)/TxPDO/input byte 1
//     PlcTask Inputs/Entradas.CA3_L9_V2_POSIC/Posicao[0] <-> Module 6 (IOL_4/4_I/O-Bytes)/TxPDO/input byte 0
//     PlcTask Inputs/Entradas.CA3_L9_V2_POSIC/Posicao[1] <-> Module 6 (IOL_4/4_I/O-Bytes)/TxPDO/input byte 1
//     PlcTask Inputs/Entradas.CA3_L9_V3_POSIC/Posicao[0] <-> Module 4 (IOL_4/4_I/O-Bytes)/TxPDO/input byte 0
//     PlcTask Inputs/Entradas.CA3_L9_V3_POSIC/Posicao[1] <-> Module 4 (IOL_4/4_I/O-Bytes)/TxPDO/input byte 1
//     PlcTask Inputs/Entradas.CA3_L9_V4_POSIC/Posicao[0] <-> Module 2 (IOL_4/4_I/O-Bytes)/TxPDO/input byte 0
//     PlcTask Inputs/Entradas.CA3_L9_V4_POSIC/Posicao[1] <-> Module 2 (IOL_4/4_I/O-Bytes)/TxPDO/input byte 1
//     PlcTask Inputs/Entradas.bPP3_L10_BD_MangRota <-> Module 7 (Digital_IN)/TxPDO/input byte 0
//     PlcTask Inputs/Entradas.bPP3_L9_BD_MangRota <-> Module 8 (Digital_IN)/TxPDO/input byte 0
//     PlcTask Inputs/ioLink.b3St1_CA3_L10_V2 <-> Module 5 (IOL_4/4_I/O-Bytes)/TxPDO/input byte 3
//     PlcTask Inputs/ioLink.b3St1_CA3_L10_V3 <-> Module 3 (IOL_4/4_I/O-Bytes)/TxPDO/input byte 3
//     PlcTask Inputs/ioLink.b3St1_CA3_L10_V4 <-> Module 1 (IOL_4/4_I/O-Bytes)/TxPDO/input byte 3
//     PlcTask Inputs/ioLink.b3St1_CA3_L9_V2 <-> Module 6 (IOL_4/4_I/O-Bytes)/TxPDO/input byte 3
//     PlcTask Inputs/ioLink.b3St1_CA3_L9_V3 <-> Module 4 (IOL_4/4_I/O-Bytes)/TxPDO/input byte 3
//     PlcTask Inputs/ioLink.b3St1_CA3_L9_V4 <-> Module 2 (IOL_4/4_I/O-Bytes)/TxPDO/input byte 3
//     PlcTask Outputs/ioLink.b0Cmd_CA3_L10_V2 <-> Module 5 (IOL_4/4_I/O-Bytes)/RxPDO/output byte 0
//     PlcTask Outputs/ioLink.b0Cmd_CA3_L10_V3 <-> Module 3 (IOL_4/4_I/O-Bytes)/RxPDO/output byte 0
//     PlcTask Outputs/ioLink.b0Cmd_CA3_L10_V4 <-> Module 1 (IOL_4/4_I/O-Bytes)/RxPDO/output byte 0
//     PlcTask Outputs/ioLink.b0Cmd_CA3_L9_V2 <-> Module 6 (IOL_4/4_I/O-Bytes)/RxPDO/output byte 0
//     PlcTask Outputs/ioLink.b0Cmd_CA3_L9_V3 <-> Module 4 (IOL_4/4_I/O-Bytes)/RxPDO/output byte 0
//     PlcTask Outputs/ioLink.b0Cmd_CA3_L9_V4 <-> Module 2 (IOL_4/4_I/O-Bytes)/RxPDO/output byte 0
//   Untitled1/Untitled1 Instance <-> Dispositivos (EtherCAT)/C1 (EK1100)/C9 (EK1122)/PU3_6 (EP3356-0022)
//     PlcTask Inputs/Entradas.PU3_WT9_bWcState <-> WcState/WcState
//     PlcTask Inputs/Entradas.PU3_WT9_rValue_REAL <-> RMB Value (Real)/Value (Real)
//     PlcTask Inputs/Entradas.PU3_WT9_stEcSlaveAmsNetAdr <-> InfoData/AdsAddr
//     PlcTask Inputs/Entradas.PU3_WT9_wState <-> InfoData/State
//     PlcTask Inputs/Entradas.PU3_WT9_wStatus <-> RMB Status/Status
//     PlcTask Outputs/Salidas.PU3_WT9_wControl <-> RMB Control/Ctrl
//   Untitled1/Untitled1 Instance <-> Dispositivos (EtherCAT)/TR_1 (EP3356-0022)
//     PlcTask Inputs/Entradas.TR_S_WT1_bWcState <-> WcState/WcState
//     PlcTask Inputs/Entradas.TR_S_WT1_rValue_REAL <-> RMB Value (Real)/Value (Real)
//     PlcTask Inputs/Entradas.TR_S_WT1_stEcSlaveAmsNetAdr <-> InfoData/AdsAddr
//     PlcTask Inputs/Entradas.TR_S_WT1_wState <-> InfoData/State
//     PlcTask Inputs/Entradas.TR_S_WT1_wStatus <-> RMB Status/Status
//     PlcTask Outputs/Salidas.TR_S_WT1_wControl <-> RMB Control/Ctrl
//   Untitled1/Untitled1 Instance <-> Dispositivos (EtherCAT)/TR_10 (EP3356-0022)
//     PlcTask Inputs/Entradas.TR_P1_WT1_bWcState <-> WcState/WcState
//     PlcTask Inputs/Entradas.TR_P1_WT1_rValue_REAL <-> RMB Value (Real)/Value (Real)
//     PlcTask Inputs/Entradas.TR_P1_WT1_stEcSlaveAmsNetAdr <-> InfoData/AdsAddr
//     PlcTask Inputs/Entradas.TR_P1_WT1_wState <-> InfoData/State
//     PlcTask Inputs/Entradas.TR_P1_WT1_wStatus <-> RMB Status/Status
//     PlcTask Outputs/Salidas.TR_P1_WT1_wControl <-> RMB Control/Ctrl
//   Untitled1/Untitled1 Instance <-> Dispositivos (EtherCAT)/TR_11 (ifm IO-Link Master AL1330)
//     PlcTask Inputs/Entradas.TR_P2_LLS <-> Module 4 (Digital_IN)/TxPDO/input byte 0
//     PlcTask Inputs/Entradas.TR_P2_ZC <-> Module 1 (Digital_IN)/TxPDO/input byte 0
//     PlcTask Inputs/Entradas.TR_P2_ZO <-> Module 2 (Digital_IN)/TxPDO/input byte 0
//     PlcTask Inputs/Entradas.TR_P2_ZS <-> Module 3 (Digital_IN)/TxPDO/input byte 0
//   Untitled1/Untitled1 Instance <-> Dispositivos (EtherCAT)/TR_12 (EP3356-0022)
//     PlcTask Inputs/Entradas.TR_P2_WT1_bWcState <-> WcState/WcState
//     PlcTask Inputs/Entradas.TR_P2_WT1_rValue_REAL <-> RMB Value (Real)/Value (Real)
//     PlcTask Inputs/Entradas.TR_P2_WT1_stEcSlaveAmsNetAdr <-> InfoData/AdsAddr
//     PlcTask Inputs/Entradas.TR_P2_WT1_wState <-> InfoData/State
//     PlcTask Inputs/Entradas.TR_P2_WT1_wStatus <-> RMB Status/Status
//     PlcTask Outputs/Salidas.TR_P2_WT1_wControl <-> RMB Control/Ctrl
//   Untitled1/Untitled1 Instance <-> Dispositivos (EtherCAT)/TR_2 (EP1908)
//     PlcTask Inputs/SafetyInputs.TR2_E1_CH01 <-> Module 1 (FSOE)/FSOE Inputs/FSOE/InputChannel1
//     PlcTask Inputs/SafetyInputs.TR2_E1_CH02 <-> Module 1 (FSOE)/FSOE Inputs/FSOE/InputChannel2
//     PlcTask Inputs/SafetyInputs.TR2_E2_CH01 <-> Module 1 (FSOE)/FSOE Inputs/FSOE/InputChannel3
//     PlcTask Inputs/SafetyInputs.TR2_E2_CH02 <-> Module 1 (FSOE)/FSOE Inputs/FSOE/InputChannel4
//     PlcTask Inputs/SafetyInputs.TR2_E3_CH01 <-> Module 1 (FSOE)/FSOE Inputs/FSOE/InputChannel5
//     PlcTask Inputs/SafetyInputs.TR2_E3_CH02 <-> Module 1 (FSOE)/FSOE Inputs/FSOE/InputChannel6
//     PlcTask Inputs/SafetyInputs.TR2_E4_CH01 <-> Module 1 (FSOE)/FSOE Inputs/FSOE/InputChannel7
//     PlcTask Inputs/SafetyInputs.TR2_E4_CH02 <-> Module 1 (FSOE)/FSOE Inputs/FSOE/InputChannel8
//   Untitled1/Untitled1 Instance <-> Dispositivos (EtherCAT)/TR_3 (EP1908)
//     PlcTask Inputs/SafetyInputs.TR3_E1_CH01 <-> Module 1 (FSOE)/FSOE Inputs/FSOE/InputChannel1
//     PlcTask Inputs/SafetyInputs.TR3_E1_CH02 <-> Module 1 (FSOE)/FSOE Inputs/FSOE/InputChannel2
//     PlcTask Inputs/SafetyInputs.TR3_E2_CH01 <-> Module 1 (FSOE)/FSOE Inputs/FSOE/InputChannel3
//     PlcTask Inputs/SafetyInputs.TR3_E2_CH02 <-> Module 1 (FSOE)/FSOE Inputs/FSOE/InputChannel4
//     PlcTask Inputs/SafetyInputs.TR3_E3_CH01 <-> Module 1 (FSOE)/FSOE Inputs/FSOE/InputChannel5
//     PlcTask Inputs/SafetyInputs.TR3_E3_CH02 <-> Module 1 (FSOE)/FSOE Inputs/FSOE/InputChannel6
//     PlcTask Inputs/SafetyInputs.TR3_E4_CH01 <-> Module 1 (FSOE)/FSOE Inputs/FSOE/InputChannel7
//     PlcTask Inputs/SafetyInputs.TR3_E4_CH02 <-> Module 1 (FSOE)/FSOE Inputs/FSOE/InputChannel8
//   Untitled1/Untitled1 Instance <-> Dispositivos (EtherCAT)/TR_4 (ifm IO-Link Master AL1332)
//     PlcTask Inputs/Entradas.TR_S_HLS <-> Module 8 (IOL_In_4Byte)/TxPDO/input byte 1
//     PlcTask Inputs/Entradas.TR_S_LLS <-> Module 7 (IOL_In_4Byte)/TxPDO/input byte 1
//     PlcTask Inputs/Entradas.TR_S_PDI <-> Module 1 (Digital_IN)/TxPDO/input byte 0
//     PlcTask Inputs/Entradas.TR_S_V2_ZC <-> Module 4 (Digital_IN)/TxPDO/input byte 0
//     PlcTask Inputs/Entradas.TR_S_V3_ZC <-> Module 2 (Digital_IN)/TxPDO/input byte 0
//     PlcTask Inputs/Entradas.TR_S_V4_ZC <-> Module 6 (Digital_IN)/TxPDO/input byte 0
//     PlcTask Inputs/Entradas.TR_S_V2_ZO <-> Module 3 (Digital_IN)/TxPDO/input byte 0
//     PlcTask Inputs/Entradas.TR_S_V4_ZO <-> Module 5 (Digital_IN)/TxPDO/input byte 0
//   Untitled1/Untitled1 Instance <-> Dispositivos (EtherCAT)/TR_5 (EX260-SEC1)
//     PlcTask Outputs/Salidas.TR_S_V1 <-> Byte 0/Output[0]
//     PlcTask Outputs/Salidas.TR_S_V2 <-> Byte 0/Output[2]
//     PlcTask Outputs/Salidas.TR_S_V3 <-> Byte 0/Output[4]
//     PlcTask Outputs/Salidas.TR_S_V4 <-> Byte 0/Output[6]
//     PlcTask Outputs/Salidas.TR_S_V5 <-> Byte 1/Output[0]
//     PlcTask Outputs/Salidas.TR_S_V6 <-> Byte 1/Output[2]
//     PlcTask Outputs/Salidas.TR_S_V7 <-> Byte 1/Output[4]
//     PlcTask Outputs/Salidas.TR_S_V8 <-> Byte 1/Output[6]
//   Untitled1/Untitled1 Instance <-> Dispositivos (EtherCAT)/TR_6 (ifm IO-Link Master AL1332)
//     PlcTask Inputs/Entradas.TR_L1_FT2_caudal/caudal[0] <-> Module 1 (IOL_16/4_I/O-Bytes)/TxPDO/input byte 5
//     PlcTask Inputs/Entradas.TR_L1_FT2_caudal/caudal[1] <-> Module 1 (IOL_16/4_I/O-Bytes)/TxPDO/input byte 4
//     PlcTask Inputs/Entradas.TR_L2_FT2_caudal/caudal[0] <-> Module 2 (IOL_16/4_I/O-Bytes)/TxPDO/input byte 5
//     PlcTask Inputs/Entradas.TR_L2_FT2_caudal/caudal[1] <-> Module 2 (IOL_16/4_I/O-Bytes)/TxPDO/input byte 4
//     PlcTask Inputs/Entradas.TR_L3_FT2_caudal/caudal[0] <-> Module 3 (IOL_16/4_I/O-Bytes)/TxPDO/input byte 5
//     PlcTask Inputs/Entradas.TR_L3_FT2_caudal/caudal[1] <-> Module 3 (IOL_16/4_I/O-Bytes)/TxPDO/input byte 4
//     PlcTask Inputs/Entradas.TR_L4_FT2_caudal/caudal[0] <-> Module 4 (IOL_16/4_I/O-Bytes)/TxPDO/input byte 5
//     PlcTask Inputs/Entradas.TR_L4_FT2_caudal/caudal[1] <-> Module 4 (IOL_16/4_I/O-Bytes)/TxPDO/input byte 4
//     PlcTask Inputs/Entradas.TR_L5_FT2_caudal/caudal[0] <-> Module 5 (IOL_16/4_I/O-Bytes)/TxPDO/input byte 5
//     PlcTask Inputs/Entradas.TR_L5_FT2_caudal/caudal[1] <-> Module 5 (IOL_16/4_I/O-Bytes)/TxPDO/input byte 4
//     PlcTask Inputs/Entradas.TR_L6_FT2_caudal/caudal[0] <-> Module 6 (IOL_16/4_I/O-Bytes)/TxPDO/input byte 5
//     PlcTask Inputs/Entradas.TR_L6_FT2_caudal/caudal[1] <-> Module 6 (IOL_16/4_I/O-Bytes)/TxPDO/input byte 4
//     PlcTask Inputs/Entradas.TR_L7_FT2_caudal/caudal[0] <-> Module 7 (IOL_16/4_I/O-Bytes)/TxPDO/input byte 5
//     PlcTask Inputs/Entradas.TR_L7_FT2_caudal/caudal[1] <-> Module 7 (IOL_16/4_I/O-Bytes)/TxPDO/input byte 4
//     PlcTask Inputs/Entradas.TR_L8_FT2_caudal/caudal[0] <-> Module 8 (IOL_16/4_I/O-Bytes)/TxPDO/input byte 5
//     PlcTask Inputs/Entradas.TR_L8_FT2_caudal/caudal[1] <-> Module 8 (IOL_16/4_I/O-Bytes)/TxPDO/input byte 4
//     PlcTask Inputs/Entradas.TR_L1_FT2_temp/temp[0] <-> Module 1 (IOL_16/4_I/O-Bytes)/TxPDO/input byte 9
//     PlcTask Inputs/Entradas.TR_L1_FT2_temp/temp[1] <-> Module 1 (IOL_16/4_I/O-Bytes)/TxPDO/input byte 8
//     PlcTask Inputs/Entradas.TR_L2_FT2_temp/temp[0] <-> Module 2 (IOL_16/4_I/O-Bytes)/TxPDO/input byte 9
//     PlcTask Inputs/Entradas.TR_L2_FT2_temp/temp[1] <-> Module 2 (IOL_16/4_I/O-Bytes)/TxPDO/input byte 8
//     PlcTask Inputs/Entradas.TR_L3_FT2_temp/temp[0] <-> Module 3 (IOL_16/4_I/O-Bytes)/TxPDO/input byte 9
//     PlcTask Inputs/Entradas.TR_L3_FT2_temp/temp[1] <-> Module 3 (IOL_16/4_I/O-Bytes)/TxPDO/input byte 8
//     PlcTask Inputs/Entradas.TR_L4_FT2_temp/temp[0] <-> Module 4 (IOL_16/4_I/O-Bytes)/TxPDO/input byte 9
//     PlcTask Inputs/Entradas.TR_L4_FT2_temp/temp[1] <-> Module 4 (IOL_16/4_I/O-Bytes)/TxPDO/input byte 8
//     PlcTask Inputs/Entradas.TR_L5_FT2_temp/temp[0] <-> Module 5 (IOL_16/4_I/O-Bytes)/TxPDO/input byte 9
//     PlcTask Inputs/Entradas.TR_L5_FT2_temp/temp[1] <-> Module 5 (IOL_16/4_I/O-Bytes)/TxPDO/input byte 8
//     PlcTask Inputs/Entradas.TR_L6_FT2_temp/temp[0] <-> Module 6 (IOL_16/4_I/O-Bytes)/TxPDO/input byte 9
//     PlcTask Inputs/Entradas.TR_L6_FT2_temp/temp[1] <-> Module 6 (IOL_16/4_I/O-Bytes)/TxPDO/input byte 8
//     PlcTask Inputs/Entradas.TR_L7_FT2_temp/temp[0] <-> Module 7 (IOL_16/4_I/O-Bytes)/TxPDO/input byte 9
//     PlcTask Inputs/Entradas.TR_L7_FT2_temp/temp[1] <-> Module 7 (IOL_16/4_I/O-Bytes)/TxPDO/input byte 8
//     PlcTask Inputs/Entradas.TR_L8_FT2_temp/temp[0] <-> Module 8 (IOL_16/4_I/O-Bytes)/TxPDO/input byte 9
//     PlcTask Inputs/Entradas.TR_L8_FT2_temp/temp[1] <-> Module 8 (IOL_16/4_I/O-Bytes)/TxPDO/input byte 8
//     PlcTask Inputs/Entradas.TR_L1_FT2_tot/total[0] <-> Module 1 (IOL_16/4_I/O-Bytes)/TxPDO/input byte 3
//     PlcTask Inputs/Entradas.TR_L1_FT2_tot/total[1] <-> Module 1 (IOL_16/4_I/O-Bytes)/TxPDO/input byte 2
//     PlcTask Inputs/Entradas.TR_L1_FT2_tot/total[2] <-> Module 1 (IOL_16/4_I/O-Bytes)/TxPDO/input byte 1
//     PlcTask Inputs/Entradas.TR_L1_FT2_tot/total[3] <-> Module 1 (IOL_16/4_I/O-Bytes)/TxPDO/input byte 0
//     PlcTask Inputs/Entradas.TR_L2_FT2_tot/total[0] <-> Module 2 (IOL_16/4_I/O-Bytes)/TxPDO/input byte 3
//     PlcTask Inputs/Entradas.TR_L2_FT2_tot/total[1] <-> Module 2 (IOL_16/4_I/O-Bytes)/TxPDO/input byte 2
//     PlcTask Inputs/Entradas.TR_L2_FT2_tot/total[2] <-> Module 2 (IOL_16/4_I/O-Bytes)/TxPDO/input byte 1
//     PlcTask Inputs/Entradas.TR_L2_FT2_tot/total[3] <-> Module 2 (IOL_16/4_I/O-Bytes)/TxPDO/input byte 0
//     PlcTask Inputs/Entradas.TR_L3_FT2_tot/total[0] <-> Module 3 (IOL_16/4_I/O-Bytes)/TxPDO/input byte 3
//     PlcTask Inputs/Entradas.TR_L3_FT2_tot/total[1] <-> Module 3 (IOL_16/4_I/O-Bytes)/TxPDO/input byte 2
//     PlcTask Inputs/Entradas.TR_L3_FT2_tot/total[2] <-> Module 3 (IOL_16/4_I/O-Bytes)/TxPDO/input byte 1
//     PlcTask Inputs/Entradas.TR_L3_FT2_tot/total[3] <-> Module 3 (IOL_16/4_I/O-Bytes)/TxPDO/input byte 0
//     PlcTask Inputs/Entradas.TR_L4_FT2_tot/total[0] <-> Module 4 (IOL_16/4_I/O-Bytes)/TxPDO/input byte 3
//     PlcTask Inputs/Entradas.TR_L4_FT2_tot/total[1] <-> Module 4 (IOL_16/4_I/O-Bytes)/TxPDO/input byte 2
//     PlcTask Inputs/Entradas.TR_L4_FT2_tot/total[2] <-> Module 4 (IOL_16/4_I/O-Bytes)/TxPDO/input byte 1
//     PlcTask Inputs/Entradas.TR_L4_FT2_tot/total[3] <-> Module 4 (IOL_16/4_I/O-Bytes)/TxPDO/input byte 0
//     PlcTask Inputs/Entradas.TR_L5_FT2_tot/total[0] <-> Module 5 (IOL_16/4_I/O-Bytes)/TxPDO/input byte 3
//     PlcTask Inputs/Entradas.TR_L5_FT2_tot/total[1] <-> Module 5 (IOL_16/4_I/O-Bytes)/TxPDO/input byte 2
//     PlcTask Inputs/Entradas.TR_L5_FT2_tot/total[2] <-> Module 5 (IOL_16/4_I/O-Bytes)/TxPDO/input byte 1
//     PlcTask Inputs/Entradas.TR_L5_FT2_tot/total[3] <-> Module 5 (IOL_16/4_I/O-Bytes)/TxPDO/input byte 0
//     PlcTask Inputs/Entradas.TR_L6_FT2_tot/total[0] <-> Module 6 (IOL_16/4_I/O-Bytes)/TxPDO/input byte 3
//     PlcTask Inputs/Entradas.TR_L6_FT2_tot/total[1] <-> Module 6 (IOL_16/4_I/O-Bytes)/TxPDO/input byte 2
//     PlcTask Inputs/Entradas.TR_L6_FT2_tot/total[2] <-> Module 6 (IOL_16/4_I/O-Bytes)/TxPDO/input byte 1
//     PlcTask Inputs/Entradas.TR_L6_FT2_tot/total[3] <-> Module 6 (IOL_16/4_I/O-Bytes)/TxPDO/input byte 0
//     PlcTask Inputs/Entradas.TR_L7_FT2_tot/total[0] <-> Module 7 (IOL_16/4_I/O-Bytes)/TxPDO/input byte 3
//     PlcTask Inputs/Entradas.TR_L7_FT2_tot/total[1] <-> Module 7 (IOL_16/4_I/O-Bytes)/TxPDO/input byte 2
//     PlcTask Inputs/Entradas.TR_L7_FT2_tot/total[2] <-> Module 7 (IOL_16/4_I/O-Bytes)/TxPDO/input byte 1
//     PlcTask Inputs/Entradas.TR_L7_FT2_tot/total[3] <-> Module 7 (IOL_16/4_I/O-Bytes)/TxPDO/input byte 0
//     PlcTask Inputs/Entradas.TR_L8_FT2_tot/total[0] <-> Module 8 (IOL_16/4_I/O-Bytes)/TxPDO/input byte 3
//     PlcTask Inputs/Entradas.TR_L8_FT2_tot/total[1] <-> Module 8 (IOL_16/4_I/O-Bytes)/TxPDO/input byte 2
//     PlcTask Inputs/Entradas.TR_L8_FT2_tot/total[2] <-> Module 8 (IOL_16/4_I/O-Bytes)/TxPDO/input byte 1
//     PlcTask Inputs/Entradas.TR_L8_FT2_tot/total[3] <-> Module 8 (IOL_16/4_I/O-Bytes)/TxPDO/input byte 0
//   Untitled1/Untitled1 Instance <-> Dispositivos (EtherCAT)/TR_7 (ifm IO-Link Master AL1330)
//     PlcTask Inputs/Entradas.TR_L10_FT2_caudal/caudal[0] <-> Module 3 (IOL_16/4_I/O-Bytes)/TxPDO/input byte 5
//     PlcTask Inputs/Entradas.TR_L10_FT2_caudal/caudal[1] <-> Module 3 (IOL_16/4_I/O-Bytes)/TxPDO/input byte 4
//     PlcTask Inputs/Entradas.TR_L11_FT2_caudal/caudal[0] <-> Module 2 (IOL_16/4_I/O-Bytes)/TxPDO/input byte 5
//     PlcTask Inputs/Entradas.TR_L11_FT2_caudal/caudal[1] <-> Module 2 (IOL_16/4_I/O-Bytes)/TxPDO/input byte 4
//     PlcTask Inputs/Entradas.TR_L12_FT2_caudal/caudal[0] <-> Module 4 (IOL_16/4_I/O-Bytes)/TxPDO/input byte 5
//     PlcTask Inputs/Entradas.TR_L12_FT2_caudal/caudal[1] <-> Module 4 (IOL_16/4_I/O-Bytes)/TxPDO/input byte 4
//     PlcTask Inputs/Entradas.TR_L9_FT2_caudal/caudal[0] <-> Module 1 (IOL_16/4_I/O-Bytes)/TxPDO/input byte 5
//     PlcTask Inputs/Entradas.TR_L9_FT2_caudal/caudal[1] <-> Module 1 (IOL_16/4_I/O-Bytes)/TxPDO/input byte 4
//     PlcTask Inputs/Entradas.TR_L10_FT2_temp/temp[0] <-> Module 3 (IOL_16/4_I/O-Bytes)/TxPDO/input byte 9
//     PlcTask Inputs/Entradas.TR_L10_FT2_temp/temp[1] <-> Module 3 (IOL_16/4_I/O-Bytes)/TxPDO/input byte 8
//     PlcTask Inputs/Entradas.TR_L11_FT2_temp/temp[0] <-> Module 2 (IOL_16/4_I/O-Bytes)/TxPDO/input byte 9
//     PlcTask Inputs/Entradas.TR_L11_FT2_temp/temp[1] <-> Module 2 (IOL_16/4_I/O-Bytes)/TxPDO/input byte 8
//     PlcTask Inputs/Entradas.TR_L12_FT2_temp/temp[0] <-> Module 4 (IOL_16/4_I/O-Bytes)/TxPDO/input byte 9
//     PlcTask Inputs/Entradas.TR_L12_FT2_temp/temp[1] <-> Module 4 (IOL_16/4_I/O-Bytes)/TxPDO/input byte 8
//     PlcTask Inputs/Entradas.TR_L9_FT2_temp/temp[0] <-> Module 1 (IOL_16/4_I/O-Bytes)/TxPDO/input byte 9
//     PlcTask Inputs/Entradas.TR_L9_FT2_temp/temp[1] <-> Module 1 (IOL_16/4_I/O-Bytes)/TxPDO/input byte 8
//     PlcTask Inputs/Entradas.TR_L10_FT2_tot/total[0] <-> Module 3 (IOL_16/4_I/O-Bytes)/TxPDO/input byte 3
//     PlcTask Inputs/Entradas.TR_L10_FT2_tot/total[1] <-> Module 3 (IOL_16/4_I/O-Bytes)/TxPDO/input byte 2
//     PlcTask Inputs/Entradas.TR_L10_FT2_tot/total[2] <-> Module 3 (IOL_16/4_I/O-Bytes)/TxPDO/input byte 1
//     PlcTask Inputs/Entradas.TR_L10_FT2_tot/total[3] <-> Module 3 (IOL_16/4_I/O-Bytes)/TxPDO/input byte 0
//     PlcTask Inputs/Entradas.TR_L11_FT2_tot/total[0] <-> Module 2 (IOL_16/4_I/O-Bytes)/TxPDO/input byte 3
//     PlcTask Inputs/Entradas.TR_L11_FT2_tot/total[1] <-> Module 2 (IOL_16/4_I/O-Bytes)/TxPDO/input byte 2
//     PlcTask Inputs/Entradas.TR_L11_FT2_tot/total[2] <-> Module 2 (IOL_16/4_I/O-Bytes)/TxPDO/input byte 1
//     PlcTask Inputs/Entradas.TR_L11_FT2_tot/total[3] <-> Module 2 (IOL_16/4_I/O-Bytes)/TxPDO/input byte 0
//     PlcTask Inputs/Entradas.TR_L12_FT2_tot/total[0] <-> Module 4 (IOL_16/4_I/O-Bytes)/TxPDO/input byte 3
//     PlcTask Inputs/Entradas.TR_L12_FT2_tot/total[1] <-> Module 4 (IOL_16/4_I/O-Bytes)/TxPDO/input byte 2
//     PlcTask Inputs/Entradas.TR_L12_FT2_tot/total[2] <-> Module 4 (IOL_16/4_I/O-Bytes)/TxPDO/input byte 1
//     PlcTask Inputs/Entradas.TR_L12_FT2_tot/total[3] <-> Module 4 (IOL_16/4_I/O-Bytes)/TxPDO/input byte 0
//     PlcTask Inputs/Entradas.TR_L9_FT2_tot/total[0] <-> Module 1 (IOL_16/4_I/O-Bytes)/TxPDO/input byte 3
//     PlcTask Inputs/Entradas.TR_L9_FT2_tot/total[1] <-> Module 1 (IOL_16/4_I/O-Bytes)/TxPDO/input byte 2
//     PlcTask Inputs/Entradas.TR_L9_FT2_tot/total[2] <-> Module 1 (IOL_16/4_I/O-Bytes)/TxPDO/input byte 1
//     PlcTask Inputs/Entradas.TR_L9_FT2_tot/total[3] <-> Module 1 (IOL_16/4_I/O-Bytes)/TxPDO/input byte 0
//   Untitled1/Untitled1 Instance <-> Dispositivos (EtherCAT)/TR_8 (ifm IO-Link Master AL1332)
//     PlcTask Inputs/Entradas.TR_L1_4_Z <-> Module 3 (Digital_IN)/TxPDO/input byte 0
//     PlcTask Inputs/Entradas.TR_L5_8_Z <-> Module 4 (Digital_IN)/TxPDO/input byte 0
//     PlcTask Inputs/Entradas.TR_L9_12_Z <-> Module 5 (Digital_IN)/TxPDO/input byte 0
//     PlcTask Inputs/Entradas.TR_S_V1_ZC <-> Module 1 (IOL_4/4_I/O-Bytes)/TxPDO/input byte 1
//     PlcTask Inputs/Entradas.TR_S_V1_ZO <-> Module 2 (IOL_4/4_I/O-Bytes)/TxPDO/input byte 1
//     PlcTask Outputs/Salidas.TR_AL1_L <-> Module 8 (IOL_4/4_I/O-Bytes)/RxPDO/output byte 1
//     PlcTask Outputs/Salidas.TR_AL2_L <-> Module 7 (IOL_4/4_I/O-Bytes)/RxPDO/output byte 1
//     PlcTask Outputs/Salidas.TR_AL2_Ac <-> Module 7 (IOL_4/4_I/O-Bytes)/RxPDO/output byte 0
//     PlcTask Outputs/Salidas.TravaHomog <-> Module 6 (Digital_OUT)/RxPDO/output byte 0
//   Untitled1/Untitled1 Instance <-> Dispositivos (EtherCAT)/TR_9 (ifm IO-Link Master AL1330)
//     PlcTask Inputs/Entradas.TR_P1_ZC <-> Module 1 (Digital_IN)/TxPDO/input byte 0
//     PlcTask Inputs/Entradas.TR_P1_ZO <-> Module 2 (Digital_IN)/TxPDO/input byte 0
//     PlcTask Inputs/Entradas.TR_P1_ZS <-> Module 3 (Digital_IN)/TxPDO/input byte 0

CONFIGURATION Untitled1
    RESOURCE PLC ON TwinCAT3
        TASK PlcTask(INTERVAL := T#10ms, PRIORITY := 6);
        PROGRAM MAIN WITH PlcTask : MAIN;
    END_RESOURCE
END_CONFIGURATION

// ---- DUTs/DUT_cfgBombas.TcDUT
TYPE DUT_cfgBombas :
STRUCT
	//Essa DUT tem os dados de configuração de cada bomba
	Apex	:INT;	//Modelo da bomba - Apex 10, apex 15, apex 20 e apex 28
	VazaoNominal	:REAL;	//Em ml/s
	Kp				:REAL;	//Parâmetro de sintonia do PID
	Ti				:REAL;	//Parametro de sintonia do PID
	BandaMorta		:REAL;	//Parâmetro de sintonia do PID
	OutMin			:REAL;	//Saída mínima do PID
	OutMax			:REAL;	//Saída máxima do PID
	PvMin			:REAL;	//Valor mínimo da variável de processo
	PvMax			:REAL;	//Valor máximo da variável de processo
END_STRUCT
END_TYPE

// ---- DUTs/DUT_cfgPosicValvula.TcDUT
TYPE DUT_cfgPosicValvula :
STRUCT
	//Essa struct estrutura os parâmetros de conversão do posicionamento das válvulas
	Aberta	:INT;
	Fechada	:INT;
END_STRUCT
END_TYPE

// ---- DUTs/DUT_PosicValvula.TcDUT
TYPE DUT_PosicValvula :
UNION
	Posicao: ARRAY[0..1] OF BYTE;
	iPosicao			:INT;
END_UNION
END_TYPE

// ---- DUTs/RecetaEdicion.TcDUT
TYPE RecetaEdicion :
STRUCT
	Nombre					:STRING;								//Nome da receita
	SetTmrHomogenizado 		:DINT := 0;								//Tempo de homogeneização
	SetTmrDescarga			:DINT := 0;								//Tempo de descarga
	SetVelocHomogenizado	:REAL := 0;								//Velocidade do homogeneizador na mistura
	SetVelocDescarga		:REAL := 0;								//Velocidade do homogeneizador na descarga
	SetCircuitosLiq			:ARRAY [1..12] OF stReceta_Circuito;	//Configuração dos liquidos
	SetCircuitosPo			:ARRAY [1..4] OF stReceta_Polvo;		//Configuração dos pós
	SetTiempoTotal			:REAL;									//Tempo total da receita
	Aspiracao				:BOOL;									//Receita com aspiração de poeira
END_STRUCT

END_TYPE

// ---- DUTs/stComboBoxRecipes.TcDUT
TYPE stComboBoxRecipes :
STRUCT
	id : INT;
	text : STRING;
	value : INT;
END_STRUCT
END_TYPE

// ---- DUTs/stListado_Liquidos.TcDUT
TYPE stListado_Liquidos :
STRUCT
	sProducto		:STRING;
	rDensidad		:REAL;// gr/ml
	iVelAspersor	:INT := 10; // 0-100%
	bAgitador		:BOOL;
	b1000s			:BOOL;
	iTempMin		:INT; // grados centigrados
	iTempMax		:INT; // grados centigrados
END_STRUCT
END_TYPE

// ---- DUTs/stListado_Polvos.TcDUT
TYPE stListado_Polvos :
STRUCT
		sProducto		:STRING:='';
		rRelacionHz		:REAL;// gr/s x  Hz
END_STRUCT
END_TYPE

// ---- DUTs/stReceta_Circuito.TcDUT
TYPE stReceta_Circuito :
STRUCT
	Paso		:INT  := 0;
	Demora		:REAL := 0;//seg
	Inyeccion	:REAL := 0;//seg
	Dosis		:REAL := 0;
END_STRUCT
END_TYPE

// ---- DUTs/stReceta_Polvo.TcDUT
TYPE stReceta_Polvo :
STRUCT
	Paso		:INT  := 0;
	Demora		:DINT := 0;//seg
	Inyeccion	:DINT := 0;//seg
	Dosis		:REAL := 0;
END_STRUCT
END_TYPE

// ---- DUTs/u_RPM.TcDUT
TYPE u_RPM :
UNION
	rpm: ARRAY[0..1] OF BYTE;
	iRpm			:INT;
END_UNION
END_TYPE

// ---- DUTs/u_SM6020.TcDUT
TYPE u_SM6020 :
UNION
	total: ARRAY[0..3] OF BYTE;
	rtotal			:REAL;// totalizado

END_UNION
END_TYPE

// ---- DUTs/u_SM6020_caudal.TcDUT
TYPE u_SM6020_caudal :
UNION
	caudal: ARRAY[0..1] OF BYTE;
	icaudal			:INT;
END_UNION
END_TYPE

// ---- DUTs/u_SM6020_temp.TcDUT
TYPE u_SM6020_temp :
UNION
	temp	:ARRAY[0..1] OF BYTE;
	itemp			:INT;
END_UNION
END_TYPE

// ---- POUs/Testes Thiago/E_State.TcDUT
{attribute 'qualified_only'}
TYPE E_State :
(
    Init,
    Idle,
    ReadOnce_CpuUsage,
    ReadOnce_CpuTemperature,
    ReadOnce_SrnMainboard,
    ReadOnce_SrnIPC,
    Write_DHCP,
    Write_IPAddr,
    ReadPeriodically,
    Error
);
END_TYPE

// ---- POUs/Testes Thiago/DUT_ConfigLavagem.TcDUT
TYPE DUT_ConfigLavagem :
STRUCT
	LavAguaLimpa:INT; //Quantidade de lavagens feitas com a água limpa
	LavAguaUsada:INT; //Quantidade de lavagens feitas com a água usada
	TempoDeCiclo:DINT; //Tempo que a bomba ficará acionada para a água chegar no fim da linha
END_STRUCT
END_TYPE

// ---- POUs/Testes Thiago/DUT_EventLogger.TcDUT
TYPE DUT_EventLogger :
STRUCT
	ID:DINT;
	Grupo:STRING;
	Data:DT;
	Hora:BYTE;
	NomeUsuario:STRING;
	Mensagem:STRING;
END_STRUCT
END_TYPE

// ---- POUs/Testes Thiago/ST_SelectStruct.TcDUT
TYPE ST_SelectStruct :
STRUCT
	ID: DINT;
	Timestamp: DT;
	Name: STRING(255);
	Value: LINT;
END_STRUCT
END_TYPE

// ---- GVL.TcGVL
{attribute 'qualified_only'}
VAR_GLOBAL
END_VAR

// ---- GVLs/CanOpen.TcGVL
{attribute 'qualified_only'}
VAR_GLOBAL
	TR_P2_WT2_rValue_REAL: REAL;
END_VAR

// ---- GVLs/Configura.TcGVL
{attribute 'qualified_only'}
VAR_GLOBAL PERSISTENT
	CantLiquidos:INT;
	CantPolvos:INT;
END_VAR

// ---- GVLs/DatosProceso.TcGVL
{attribute 'qualified_only'}
VAR_GLOBAL PERSISTENT
	CargarLote		:BOOL;		//Carrega lote
	Kg_a_Procesar	:REAL;		//Quantidade total de semente a ser tratada
	NomeLote		:STRING;	//Nome ou número do lote
	LoteCargado		:BOOL;		//Lote carregado
	KgLote_Procesados	:REAL;	//Quantidade de semente tratada
	ConsumoCircuito_1	:REAL;	//Consumo de liquido do circuito 1
	ConsumoCircuito_2	:REAL;	//Consumo de liquido do circuito 2
	ConsumoCircuito_3	:REAL;	//Consumo de liquido do circuito 3
	ConsumoCircuito_4	:REAL;	//Consumo de liquido do circuito 4
	ConsumoCircuito_5	:REAL;	//Consumo de liquido do circuito 5
	ConsumoCircuito_6	:REAL;	//Consumo de liquido do circuito 6
	ConsumoCircuito_7	:REAL;	//Consumo de liquido do circuito 7
	ConsumoCircuito_8	:REAL;	//Consumo de liquido do circuito 8
	ConsumoCircuito_9	:REAL;	//Consumo de liquido do circuito 9
	ConsumoCircuito_10	:REAL;	//Consumo de liquido do circuito 10
	ConsumoCircuito_11	:REAL;	//Consumo de liquido do circuito 11
	ConsumoCircuito_12	:REAL;	//Consumo de liquido do circuito 12
	ConsumoPolvo_1		:REAL;	//Consumo de pó 1
	ConsumoPolvo_2		:REAL;	//Consumo de pó 2 
	TempoRestante		:REAL;	//Aproximação do tempo restante para tratar toda a semente do lote
	TempoTratamento		:UDINT;	//Tempo decorrido do tratamento atual
	TempoTotal			:REAL;	//Tempo total do tratamento
	InicioTratamento	:UDINT;	//DAta e hora do inicio do tratamento atual
	
END_VAR

// ---- GVLs/Entradas.TcGVL
{attribute 'qualified_only'}
VAR_GLOBAL
	//
	Pulsador_emerg 	AT %I* :BOOL;
	ReposicionEmerg AT %I* :BOOL;
	TR_S_PDI		AT %I* :BOOL;//presion aire ok
	
	//Agitadores
	bPP1_L1_AG_Z	AT%I* :BOOL;
	bPP1_L2_AG_Z	AT%I* :BOOL;
	bPP1_L3_AG_Z	AT%I* :BOOL;
	bPP1_L4_AG_Z	AT%I* :BOOL;
	bPP2_L5_AG_Z	AT%I* :BOOL;
	bPP2_L6_AG_Z	AT%I* :BOOL;
	bPP2_L7_AG_Z	AT%I* :BOOL;
	bPP2_L8_AG_Z	AT%I* :BOOL;
	bPP3_L9_AG_Z	AT%I* :BOOL;
	bPP3_L10_AG_Z	AT%I* :BOOL;
	bPP3_L11_AG_Z	AT%I* :BOOL;
	bPP3_L12_AG_Z	AT%I* :BOOL;
	//Soplador tratadora
	bTR_S_VE1_Z AT%I* :BOOL;
	
	//Lavado
	bHLS_TkAguaResidual:BOOL;
	
	//TR_S_WT1 semilla
	TR_S_WT1_wStatus AT %I*:WORD;
	TR_S_WT1_rValue_REAL AT %I*:REAL;
	TR_S_WT1_nValue_DINT AT %I* :DINT;
	TR_S_WT1_nValue_Supply AT %I*:DINT;		(*only for voltage measurement, change PDO settings"*)
	TR_S_WT1_nValue_Bridge AT %I*:DINT;		(*only for voltage measurement, change PDO settings"*)
	TR_S_WT1_stEcSlaveAmsNetAdr AT %I* :ST_AmsAddr;
	TR_S_WT1_bWcState AT %I*:BOOL;
	TR_S_WT1_wState AT %I*:WORD;
	
	//Tratadora
	TR_S_V1_ZC AT%I* :BOOL;
	TR_S_V1_ZO AT%I* :BOOL;
	TR_S_V2_ZC AT%I* :BOOL;//corte grueso cerrado
	TR_S_V2_ZO AT%I* :BOOL;//corte grueso abierto
	TR_S_V3_ZC AT%I* :BOOL;//corte fino cerrado
	TR_S_V3_ZO AT%I* :BOOL;
	TR_S_V4_ZC AT%I* :BOOL;//descarga balanza cerrada
	TR_S_V4_ZO AT%I* :BOOL;//descarga balanza abierta
	TR_S_LLS AT%I* :BOOL;//nivel minimo tolva descarga semilla
	TR_S_HLS AT%I* :BOOL;//nivel maximo tolva descarga semilla
	
	TR_L1_4_Z AT%I* :BOOL;//inyector L1 a L4 en posicion
	TR_L5_8_Z AT%I* :BOOL;//inyector L5 a L8 en posicion
	TR_L9_12_Z AT%I* :BOOL;//inyector L9 a L12 en posicion
	
	wTR_S_VF1_St AT%I* :WORD;//homoogenizador
	wTR_S_VF1_PV AT%I* :WORD;//homoogenizador
	wTR_S_VF2_St AT%I* :WORD;//aspersor
	wTR_S_VF2_PV AT%I* :WORD;//aspersor
	
	//Bomba Circuito 1
	wPP1_L1_BD_St AT%I* :WORD;
	wPP1_L1_BD_PV AT%I* :WORD;
	bPP1_L1_BD_MangRota AT%I* :BOOL;
	//Bomba Circuito 2
	wPP1_L2_BD_St AT%I* :WORD;
	wPP1_L2_BD_PV AT%I* :WORD;
	bPP1_L2_BD_MangRota AT%I* :BOOL;
	//Bomba Circuito 3
	wPP1_L3_BD_St AT%I* :WORD;
	wPP1_L3_BD_PV AT%I* :WORD;
	bPP1_L3_BD_MangRota AT%I* :BOOL;
	//Bomba Circuito 4
	wPP1_L4_BD_St AT%I* :WORD;
	wPP1_L4_BD_PV AT%I* :WORD;
	bPP1_L4_BD_MangRota AT%I* :BOOL;
	//Bomba Circuito 5
	wPP2_L5_BD_St AT%I* :WORD;
	wPP2_L5_BD_PV AT%I* :WORD;
	bPP2_L5_BD_MangRota AT%I* :BOOL;
	//Bomba Circuito 6
	wPP2_L6_BD_St AT%I* :WORD;
	wPP2_L6_BD_PV AT%I* :WORD;
	bPP2_L6_BD_MangRota AT%I* :BOOL;
	//Bomba Circuito 7
	wPP2_L7_BD_St AT%I* :WORD;
	wPP2_L7_BD_PV AT%I* :WORD;
	bPP2_L7_BD_MangRota AT%I* :BOOL;
	//Bomba Circuito 8
	wPP2_L8_BD_St AT%I* :WORD;
	wPP2_L8_BD_PV AT%I* :WORD;
	bPP2_L8_BD_MangRota AT%I* :BOOL;
	//Bomba Circuito 9
	wPP3_L9_BD_St AT%I* :WORD;
	wPP3_L9_BD_PV AT%I* :WORD;
	bPP3_L9_BD_MangRota AT%I* :BOOL;
	//Bomba Circuito 10
	wPP3_L10_BD_St AT%I* :WORD;
	wPP3_L10_BD_PV AT%I* :WORD;
	bPP3_L10_BD_MangRota AT%I* :BOOL;
	//Bomba Circuito 11
	wPP3_L11_BD_St AT%I* :WORD;
	wPP3_L11_BD_PV AT%I* :WORD;
	bPP3_L11_BD_MangRota AT%I* :BOOL;
	//Bomba Circuito 12
	wPP3_L12_BD_St AT%I* :WORD;
	wPP3_L12_BD_PV AT%I* :WORD;
	bPP3_L12_BD_MangRota AT%I* :BOOL;
	
	//Caudalimetro Calibracion
	CA1_L1_FT1_tot AT%I* :u_SM6020;
	CA1_L1_FT1_temp AT%I* :u_SM6020_temp;
	CA1_L1_FT1_caudal AT%I* :u_SM6020_caudal;
	CA1_L2_FT1_tot AT%I* :u_SM6020;
	CA1_L2_FT1_temp AT%I* :u_SM6020_temp;
	CA1_L2_FT1_caudal AT%I* :u_SM6020_caudal;
	CA1_L3_FT1_Tot AT%I* :u_SM6020;
	CA1_L3_FT1_temp AT%I* :u_SM6020_temp;
	CA1_L3_FT1_caudal AT%I* :u_SM6020_caudal;
	CA1_L4_FT1_tot AT%I* :u_SM6020;
	CA1_L4_FT1_temp AT%I* :u_SM6020_temp;
	CA1_L4_FT1_caudal AT%I* :u_SM6020_caudal;
	CA2_L5_FT1_tot AT%I* :u_SM6020;
	CA2_L5_FT1_temp AT%I* :u_SM6020_temp;
	CA2_L5_FT1_caudal AT%I* :u_SM6020_caudal;
	CA2_L6_FT1_tot AT%I* :u_SM6020;
	CA2_L6_FT1_temp AT%I* :u_SM6020_temp;
	CA2_L6_FT1_caudal AT%I* :u_SM6020_caudal;
	CA2_L7_FT1_tot AT%I* :u_SM6020;
	CA2_L7_FT1_temp AT%I* :u_SM6020_temp;
	CA2_L7_FT1_caudal AT%I* :u_SM6020_caudal;
	CA2_L8_FT1_tot AT%I* :u_SM6020;
	CA2_L8_FT1_temp AT%I* :u_SM6020_temp;
	CA2_L8_FT1_caudal AT%I* :u_SM6020_caudal;
	CA3_L9_FT1_tot AT%I* :u_SM6020;
	CA3_L9_FT1_temp AT%I* :u_SM6020_temp;
	CA3_L9_FT1_caudal AT%I* :u_SM6020_caudal;
	CA3_L10_FT1_tot AT%I* :u_SM6020;
	CA3_L10_FT1_temp AT%I* :u_SM6020_temp;
	CA3_L10_FT1_caudal AT%I* :u_SM6020_caudal;
	CA3_L11_FT1_tot AT%I* :u_SM6020;
	CA3_L11_FT1_temp AT%I* :u_SM6020_temp;
	CA3_L11_FT1_caudal AT%I* :u_SM6020_caudal;
	CA3_L12_FT1_tot AT%I* :u_SM6020;
	CA3_L12_FT1_temp AT%I* :u_SM6020_temp;
	CA3_L12_FT1_caudal AT%I* :u_SM6020_caudal;
	
	//Caudalimetro Tratadora
	TR_L1_FT2_tot AT%I* :u_SM6020;
	TR_L1_FT2_temp AT%I* :u_SM6020_temp;
	TR_L1_FT2_caudal AT%I* :u_SM6020_caudal;
	TR_L2_FT2_tot AT%I* :u_SM6020;
	TR_L2_FT2_temp AT%I* :u_SM6020_temp;
	TR_L2_FT2_caudal AT%I* :u_SM6020_caudal;
	TR_L3_FT2_tot AT%I* :u_SM6020;
	TR_L3_FT2_temp AT%I* :u_SM6020_temp;
	TR_L3_FT2_caudal AT%I* :u_SM6020_caudal;
	TR_L4_FT2_tot AT%I* :u_SM6020;
	TR_L4_FT2_temp AT%I* :u_SM6020_temp;
	TR_L4_FT2_caudal AT%I* :u_SM6020_caudal;
	TR_L5_FT2_tot AT%I* :u_SM6020;
	TR_L5_FT2_temp AT%I* :u_SM6020_temp;
	TR_L5_FT2_caudal AT%I* :u_SM6020_caudal;
	TR_L6_FT2_tot AT%I* :u_SM6020;
	TR_L6_FT2_temp AT%I* :u_SM6020_temp;
	TR_L6_FT2_caudal AT%I* :u_SM6020_caudal;
	TR_L7_FT2_tot AT%I* :u_SM6020;
	TR_L7_FT2_temp AT%I* :u_SM6020_temp;
	TR_L7_FT2_caudal AT%I* :u_SM6020_caudal;
	TR_L8_FT2_tot AT%I* :u_SM6020;
	TR_L8_FT2_temp AT%I* :u_SM6020_temp;
	TR_L8_FT2_caudal AT%I* :u_SM6020_caudal;
	TR_L9_FT2_tot AT%I* :u_SM6020;
	TR_L9_FT2_temp AT%I* :u_SM6020_temp;
	TR_L9_FT2_caudal AT%I* :u_SM6020_caudal;
	TR_L10_FT2_tot AT%I* :u_SM6020;
	TR_L10_FT2_temp AT%I* :u_SM6020_temp;
	TR_L10_FT2_caudal AT%I* :u_SM6020_caudal;
	TR_L11_FT2_tot AT%I* :u_SM6020;
	TR_L11_FT2_temp AT%I* :u_SM6020_temp;
	TR_L11_FT2_caudal AT%I* :u_SM6020_caudal;
	TR_L12_FT2_tot AT%I* :u_SM6020;
	TR_L12_FT2_temp AT%I* :u_SM6020_temp;
	TR_L12_FT2_caudal AT%I* :u_SM6020_caudal;	
	
	//Balanza probeta CA1
	CA1_WT1_wStatus AT%I* :WORD;
	CA1_WT1_rValue_REAL AT %I*:REAL;
	CA1_WT1_nValue_DINT AT %I* :DINT;
	CA1_WT1_stEcSlaveAmsNetAdr AT%I* :ST_AmsAddr;
	CA1_WT1_bWcState  AT%I* :BOOL;
	CA1_WT1_wState  AT%I*:WORD;
	//Balanza probeta CA2
	CA2_WT1_wStatus AT%I* :WORD;
	CA2_WT1_rValue_REAL AT %I*:REAL;
	CA2_WT1_nValue_DINT  :DINT;
	CA2_WT1_stEcSlaveAmsNetAdr AT%I* :ST_AmsAddr;
	CA2_WT1_bWcState  AT%I* :BOOL;
	CA2_WT1_wState  AT%I*:WORD;
	//Balanza probeta CA3
	CA3_WT1_wStatus AT%I* :WORD;
	CA3_WT1_rValue_REAL AT %I*:REAL;
	CA3_WT1_nValue_DINT  :DINT;
	CA3_WT1_stEcSlaveAmsNetAdr AT%I* :ST_AmsAddr;
	CA3_WT1_bWcState  AT%I* :BOOL;
	CA3_WT1_wState  AT%I*:WORD;
	//Balanza IBC 1
	PU1_WT1_wStatus AT%I* :WORD;
	PU1_WT1_rValue_REAL AT %I*:REAL;
	PU1_WT1_nValue_DINT  :DINT;
	PU1_WT1_stEcSlaveAmsNetAdr AT%I* :ST_AmsAddr;
	PU1_WT1_bWcState  AT%I* :BOOL;
	PU1_WT1_wState  AT%I*:WORD;
	//Balanza IBC 2
	PU1_WT2_wStatus AT%I* :WORD;
	PU1_WT2_rValue_REAL AT %I*:REAL;
	PU1_WT2_nValue_DINT  :DINT;
	PU1_WT2_stEcSlaveAmsNetAdr AT%I* :ST_AmsAddr;
	PU1_WT2_bWcState  AT%I* :BOOL;
	PU1_WT2_wState  AT%I*:WORD;
	//Balanza IBC 3
	PU1_WT3_wStatus AT%I* :WORD;
	PU1_WT3_rValue_REAL AT %I*:REAL;
	PU1_WT3_nValue_DINT  :DINT;
	PU1_WT3_stEcSlaveAmsNetAdr AT%I* :ST_AmsAddr;
	PU1_WT3_bWcState  AT%I* :BOOL;
	PU1_WT3_wState  AT%I*:WORD;
	//Balanza IBC 4
	PU1_WT4_wStatus AT%I* :WORD;
	PU1_WT4_rValue_REAL AT %I*:REAL;
	PU1_WT4_nValue_DINT  :DINT;
	PU1_WT4_stEcSlaveAmsNetAdr AT%I* :ST_AmsAddr;
	PU1_WT4_bWcState  AT%I* :BOOL;
	PU1_WT4_wState  AT%I*:WORD;
	//Balanza IBC 5
	PU2_WT5_wStatus AT%I* :WORD;
	PU2_WT5_rValue_REAL AT %I*:REAL;
	PU2_WT5_nValue_DINT  :DINT;
	PU2_WT5_stEcSlaveAmsNetAdr AT%I* :ST_AmsAddr;
	PU2_WT5_bWcState  AT%I* :BOOL;
	PU2_WT5_wState  AT%I*:WORD;
	//Balanza IBC 6
	PU2_WT6_wStatus AT%I* :WORD;
	PU2_WT6_rValue_REAL AT %I*:REAL;
	PU2_WT6_nValue_DINT  :DINT;
	PU2_WT6_stEcSlaveAmsNetAdr AT%I* :ST_AmsAddr;
	PU2_WT6_bWcState  AT%I* :BOOL;
	PU2_WT6_wState  AT%I*:WORD;
	//Balanza IBC 7
	PU2_WT7_wStatus AT%I* :WORD;
	PU2_WT7_rValue_REAL AT %I*:REAL;
	PU2_WT7_nValue_DINT  :DINT;
	PU2_WT7_stEcSlaveAmsNetAdr AT%I* :ST_AmsAddr;
	PU2_WT7_bWcState  AT%I* :BOOL;
	PU2_WT7_wState  AT%I*:WORD;
	//Balanza IBC 8
	PU2_WT8_wStatus AT%I* :WORD;
	PU2_WT8_rValue_REAL AT %I*:REAL;
	PU2_WT8_nValue_DINT  :DINT;
	PU2_WT8_stEcSlaveAmsNetAdr AT%I* :ST_AmsAddr;
	PU2_WT8_bWcState  AT%I* :BOOL;
	PU2_WT8_wState  AT%I*:WORD;
	//Balanza IBC 9
	PU3_WT9_wStatus AT%I* :WORD;
	PU3_WT9_rValue_REAL AT %I*:REAL;
	PU3_WT9_nValue_DINT  :DINT;
	PU3_WT9_stEcSlaveAmsNetAdr AT%I* :ST_AmsAddr;
	PU3_WT9_bWcState  AT%I* :BOOL;
	PU3_WT9_wState  AT%I*:WORD;
	//Balanza IBC 10
	PU3_WT10_wStatus AT%I* :WORD;
	PU3_WT10_rValue_REAL AT %I*:REAL;
	PU3_WT10_nValue_DINT  :DINT;
	PU3_WT10_stEcSlaveAmsNetAdr AT%I* :ST_AmsAddr;
	PU3_WT10_bWcState  AT%I* :BOOL;
	PU3_WT10_wState  AT%I*:WORD;
	//Balanza IBC 11
	PU3_WT11_wStatus AT%I* :WORD;
	PU3_WT11_rValue_REAL AT %I*:REAL;
	PU3_WT11_nValue_DINT  :DINT;
	PU3_WT11_stEcSlaveAmsNetAdr AT%I* :ST_AmsAddr;
	PU3_WT11_bWcState  AT%I* :BOOL;
	PU3_WT11_wState  AT%I*:WORD;
	//Balanza IBC 12
	PU3_WT12_wStatus AT%I* :WORD;
	PU3_WT12_rValue_REAL AT %I*:REAL;
	PU3_WT12_nValue_DINT  :DINT;
	PU3_WT12_stEcSlaveAmsNetAdr AT%I* :ST_AmsAddr;
	PU3_WT12_bWcState  AT%I* :BOOL;
	PU3_WT12_wState  AT%I*:WORD;
	//Balanza Polvo 1
	TR_P1_WT1_wStatus AT%I* :WORD;
	TR_P1_WT1_rValue_REAL AT %I*:REAL;
	TR_P1_WT1_nValue_DINT  :DINT;
	TR_P1_WT1_stEcSlaveAmsNetAdr AT%I* :ST_AmsAddr;
	TR_P1_WT1_bWcState  AT%I* :BOOL;
	TR_P1_WT1_wState  AT%I*:WORD;
	//Balanza Polvo 2
	TR_P2_WT1_wStatus AT%I* :WORD;
	TR_P2_WT1_rValue_REAL AT %I*:REAL;
	TR_P2_WT1_nValue_DINT  :DINT;
	TR_P2_WT1_stEcSlaveAmsNetAdr AT%I* :ST_AmsAddr;
	TR_P2_WT1_bWcState  AT%I* :BOOL;
	TR_P2_WT1_wState  AT%I*:WORD;
	//Dosificador Polvo 1
	TR_P1_VF_St AT%I* :WORD;
	TR_P1_VF_PV AT%I* :WORD;
	//Dosificador Polvo 2
	TR_P2_VF_St AT%I* :WORD;
	TR_P2_VF_PV AT%I* :WORD;
	//Vibrador  Polvo 1
	TR_P1_VI_St AT%I* :WORD;
	TR_P1_VI_PV AT%I* :WORD;
	// Vibrador  Polvo 2
	TR_P2_VI_St AT%I* :WORD;
	TR_P2_VI_PV AT%I* :WORD;
	
	TR_P1_ZS	AT %I* :BOOL;	//sensor velocidad dosif Polvo 1
	TR_P1_ZC	AT %I* :BOOL;	//posicion dosificar Polvo 1
	TR_P1_ZO	AT %I* :BOOL;	//posicion calibrar Polvo 1
	TR_P1_LLS	AT %I* :BOOL;	// nivel minimo Polvo 1
	TR_P2_ZS	AT %I* :BOOL;	//sensor velocidad dosif Polvo 2	
	TR_P2_ZC	AT %I* :BOOL;	//posicion dosificar Polvo 2
	TR_P2_ZO	AT %I* :BOOL;	//posicion calibrar Polvo 2
	TR_P2_LLS	AT %I* :BOOL;	// nivel minimo Polvo 2	
	
	//Perifericos Elevador 1
	wPE_B_VF1_St AT%I* :WORD;
	wPE_B_VF1_PV AT%I* :WORD;
	
	//Perifericos Elevador 2
	wPE_H_VF1_St AT%I* :WORD;
	wPE_H_VF1_PV AT%I* :WORD;
	
	//Perifericos Elevador 3
	wPE_H_VF2_St AT%I* :WORD;
	wPE_H_VF2_PV AT%I* :WORD;
	
	PE_B1_V1_ZO			AT%I* :BOOL;	//descarga intermedia 1 no descarga
	PE_B2_V1_ZO			AT%I* :BOOL;	//descarga intermedia 2 no descarga
	PE_B3_V1_ZO			AT%I* :BOOL;	//descarga intermedia 3 no descarga	
	PE_B1_LLS			AT%I* :BOOL;	//nivel minimo tolva embolse CE1	
	PE_B2_LLS			AT%I* :BOOL;	//nivel minimo tolva embolse CE2
	PE_B3_LLS			AT%I* :BOOL;	//nivel minimo tolva embolse CE3
	PE_B1_HLS			AT%I* :BOOL;	//nivel maximo tolva embolse CE1	
	PE_B2_HLS			AT%I* :BOOL;	//nivel maximo tolva embolse CE2
	PE_B3_HLS			AT%I* :BOOL;	//nivel maximo tolva embolse CE3
	PE_H_HLS			AT%I* :BOOL;	//nivel maximo tolva 30t
	TR_CDT_LLS			AT%I* :BOOL;	//nivel trabajo descarga tratadora	
	
